FUNCTION_BLOCK "FU SEW DFE32B - PN_REL"	// FB 6119
TITLE = Control of SEW frequency converter with DFE32B via Profinet
//Building:
//Date         Editor                                                     Version
//--------------------------------------------------------------------------------
//31.08.10     A.Kremer (kal)                                            01.00.00
//
//Modifications:
//No. Date     Edit  Description                                    Index Version
//--------------------------------------------------------------------------------
//01  24.04.12 sra   Anpassung zur Integration als Standardbaustein (001) 01.01.00
//02  23.11.15 kst   Anpassung allgemein                            (002) 01.02.00
//03  17.02.16 sra   out_FB_Fehlermeldung = INT                     (003) 01.02.01
//________________________________________________________________________________
//Functional description:
//
//The function cummunicates to a SEW frequency converter MOVITRAC B via Profinet
//interface DFE32B.
//
//Hardwareconfiguration:
//Install GSDML file in hardware catalogue:
// GSDML-V2.1-SEW-DFE-DFS-2Ports-20070426.xml (Internet: www.SEW-EURODRIVE.de)
//
//After the installation you can find the Profinet module  "SEW Gateway DFE32B 
//V1.2" in the hardware catalogue under the menu: "Profinet IO -> other FIELD 
//DEVICES -> Drives -> SEW -> DFE/DFS (2Ports) ->"
//
//Insert this module to the hardware and configurate the following module
//     Slot 1: Empty
//from Slot 2: AS 1 Antrieb (1x3PD)   as often as the number of freq.converter    
// 
//
//
//!!! The nominal motor frequency, motor speed and the nominal motor current must 
//    be transferred to ensure the block functions correctly.
//
//
//Settings at DFE32B:
//
//1. Set IP address via Software: 
//
//2. Execute auto setup at DFE32B by setting DIP switch 2 (AS) to ON
//   All FCs must be switched on and the SBus address set
//   With the auto setup function (DIP switch "AS") it is possible to set up 
//   DFE32B as the gateway without a PC. The function is executed once when the 
//   DIP switch is switched on. The DIP switch must then remain on. The function 
//   can be executed again by switching the DIP switch off and on again.
//
//Frequency converter settings
//
//1. P100 Set setpoint source to SBUS -> value = 10
//
//2. P101 Set control source to SBus -> value 3
//
//3. P301 Set minimum speed in rpm (master value = 15)
//
//4. P302 Set maximum speed in rpm (factory setting = 1500)
//
//5. P303 Set current limit (in % of FC nominal current)
//   (Factory setting =150%)
//
//6. P320 Set automatic motor matching to on (standard setting)
//   (to gauge the motor at start)
//
//7. P500 Switch on speed monitoring
//   (in the case of fault messages P501 increase speed monitoring delay time)
//
//8. P601, P603 and P608 Set binary inputs to ""no function" (=0)
//   Set P602 to 1 = enable (factory setting) DI03 must be bypassed
//
//9. P604 for operation with PTC resistor set to 26 (TF message) otherwise
//   .... zeroing.
//   
//11. P881 Set SBus address of respective frequency converter (from 1 in
//    ascending order)
//
//12. P883 Bus monitoring time -> 5 [s]
//
//13. P884 Check SBus baud rate -> value 500/500 kBaud
//
//14. P870-P872 Setpoint description PA1-PA3
//       P870 = control word 1
//       P871 = speed
//       P872 = reserve
//    P873-P876 Actual value description PE1-PE3
//       P873 = status word 1
//       P874 = speed
//       P875 = output current in % of nominal current
//
AUTHOR : kal
FAMILY : AZO
NAME : standard
VERSION : 0.0
VAR_INPUT
  in_PEA_Adresse : INT ;	//Basisadresse für EA-Daten im PEA-Bereich
  in_FU_Nummer : INT ;	//FU Nummer zur Berechnung des Offsets der Peripherie-EAs
  in_Motordaten_J_N : BOOL ;	//nicht möglich => CLR
  in_Freigabe : BOOL ;	//Steuersignal 1 setzen zum Starten des FUs
  in_Linkslauf : BOOL ;	//Frequenzumformer Linkslauf ein
  in_Quittierung_Stoerung : BOOL ;	//Störung quittieren
  in_Sollfrequenz : REAL ;	//Sollfrequenz in Hz
  in_Motorleistungsfaktor : REAL ;	//nicht vorhanden => 0
  in_Motornennfrequenz : REAL ;	//Wertebereich: 0 - 100 Hz
  in_Motornenndrehzahl : REAL ;	//Wertebereich: 0 - 10000 U/min
  in_Motornennstrom : REAL ;	//Wertebereich: 0- ... A
  in_Motornennspannung : REAL ;	//nicht vorhanden => 0
  in_Motornennleistung : REAL ;	//nicht vorhanden => 0
END_VAR
VAR_OUTPUT
  out_Istfrequenz : REAL ;	//Istfrequenz in Hz
  out_Istdrehzahl : REAL ;	//Istdrehzahl in U/min
  out_Leistung : REAL ;	//nicht vorhanden => 0
  out_Drehmoment : REAL ;	//nicht vorhanden => 0
  out_Motorspannung : REAL ;	//nicht vorhanden => 0
  out_Ausgangsstrom : REAL ;	//Ausgangsstrom des FU
  out_Stoerung : BOOL ;	//1=Gerätestörung
  out_Warnung : BOOL ;
  out_Sollwert_erreicht : BOOL ;	//zeigt 1 an, wenn Istwert gleich Sollwert ist
  out_laeuft : BOOL ;	//=1 wenn Istdrehzahl > 0
  out_FB_Fehlermeldung : INT ;	//0 = ok ; sonst Fehler_Code_L2Dp
  out_Stoerungsnummer : DINT ;	//Stoerungsnummer, bzw. Betriebszustand wenn keine Störung aktiv
END_VAR
VAR
  reserve : ARRAY  [58 .. 99 ] OF BYTE ;
  Prozessdatenkanal_in : STRUCT 	//Prozesseingangsdaten
   PI1_Statuswort : STRUCT
    Zustand_Fehlercode : BYTE ;
    Endstufe_freigegeben : BOOL ;
    Umrichter_betriebsbereit : BOOL ;
    PA_Daten_freigegeben : BOOL ;
    reserve_3 : BOOL ;
    reserve_4 : BOOL ;
    Stoerung_Warnung : BOOL ;
    reserve_6 : BOOL ;	//0 = 1. Satz; 1 = 2. Satz
    reserve_7 : BOOL ;	//0 = 1. Satz; 1 = 2. Satz
   END_STRUCT ;
   PI2_Istdrehzahl : INT ;
   PI3_Ausgangsstrom : INT ;
  END_STRUCT ;
  Prozessdatenkanal_out : STRUCT 	//Prozessausgangsdaten
   PO1_Steuerwort : STRUCT
    Drehrichtung : BOOL ;	//0 = rechts; 1 = links
    Motorpoti_auf : BOOL ;	//00=11= keine Änderung; 01=Hochlauf, 02=Tieflauf
    Motorpoti_ab : BOOL ;
    Festsollwerte_0 : BOOL ;	//00 = Feldbus
    Festsollwerte_1 : BOOL ;
    Festsollwert_Umschaltung : BOOL ;
    reserve_14 : BOOL ;
    reserve_15 : BOOL ;
    Reglersperre : BOOL ;	//Freigabe = '110', sonst Halt
    Freigabe_Schnellstop : BOOL ;
    Freigabe_Normalhalt : BOOL ;
    reserve_3 : BOOL ;
    reserve_4 : BOOL ;
    reserve_5 : BOOL ;	//0 = 1.Satz; 1 = 2.Satz
    Reset_Stoerung : BOOL ;	//0 = 1.Satz; 1 = 2.Satz
    reserve_7 : BOOL ;
   END_STRUCT ;
   PO2_Solldrehzahl : INT ;	//in %
   PO3_keine_Fkt : INT ;
  END_STRUCT ;
  Datenuebertragung : STRUCT
   Schritt_aktiv : BOOL ;
  END_STRUCT ;
  reserve_1 : ARRAY  [122 .. 137 ] OF BYTE ;
END_VAR
VAR_TEMP
  IO_Adr_Parameterkanal : WORD ;
  IO_Adr_Prozessdatenkanal : WORD ;
  Ret_Val_SFC14_1 : INT ;
  Ret_Val_SFC14_2 : INT ;
  Ret_Val_SFC15_1 : INT ;
  Ret_Val_SFC15_2 : INT ;
  SimFactor : REAL ;	//(001)
  Solldrehzahl_tmp : REAL ;
END_VAR
BEGIN
NETWORK
TITLE = Bausteinende wenn PEA-Adresse = 0
      L     #in_PEA_Adresse;
      L     0;
      ==I;
      BEC;
NETWORK
TITLE = Simulation
//Über die Simulaitonsmerker "M 0.5 Simulation intern" oder "M 0.6 Simulation 
//AVP" 
//wird die Funktion des FUs simuliert:
//- Fehler werden zurückgesetzt
//- Bei Freigabe Istdrehzahl=Solldrehzahl, Betrieb und Solldrehzahl erreicht = 
//True
//(002) Überarbeitung 
      O     "M0.5 SimulationInternal";
      O     "M0.6 SimulationAVP";
      JCN   NSIM;
// <<(002)
      SET;
      R     #out_Stoerung;
      R     #out_Warnung;
// >>(002)
      L     L#0;
      T     #out_Stoerungsnummer;
      A     #in_Freigabe;
      =     #out_laeuft;
      =     #out_Sollwert_erreicht;
      L     #in_Sollfrequenz;
      JC    SIMD;
      L     0.000000e+00;
SIMD: T     #out_Istfrequenz;
// <<(002)
// Faktor berechnen
//     L     #out_Istfrequenz
//     L     #in_Motornennfrequenz
//      /R    
//     T     #SimFactor
// Istdrehzahl
//     L     #in_Motornenndrehzahl
//     L     #SimFactor
//      *R    
//     T     #out_Istdrehzahl
// Istleistung
//     L     #in_Motornennleistung
//     L     #SimFactor
//      *R    
//     T     #out_Leistung
// Istspannung
//     L     #in_Motornennspannung
//     L     #SimFactor
//      *R    
//     T     #out_Motorspannung
// Iststrom
//     L     #in_Motornennstrom
//     L     #SimFactor
//      *R    
//     T     #out_Ausgangsstrom
// >>(002)
      BEU;
NSIM: NOP   0;
NETWORK
TITLE = Daten von FU einlesen
//FU-Daten auslesen mit SFC14
//PEA_Adresse zeigt auf den Anfang des EA-Bereiches.
// 6-Byte Prozessdatenkanal
// <<(002)
      L     #in_FU_Nummer;
      +     -1;
      L     6;	// Länge eines Parameterkanals je FU
      *I;
      L     #in_PEA_Adresse;
      +I;
      T     #IO_Adr_Prozessdatenkanal;	// Daten des jeweiligen FU = PEA-Adresse + 8 Byte + (FU-Nr. - 1) * 6
// >>(002)
      CALL  "DPRD_DAT" (
           LADDR                    := #IO_Adr_Prozessdatenkanal,
           RET_VAL                  := #Ret_Val_SFC14_2,
           RECORD                   := #Prozessdatenkanal_in);
NETWORK
TITLE = Istdrehzahl auswerten
//Istdrehzahl in 0,2 U/min
      L     #Prozessdatenkanal_in.PI2_Istdrehzahl;
      ITD;
      DTR;
      L     5.000000e+00;
      /R;
      T     #out_Istdrehzahl;
NETWORK
TITLE = Istfrequenz auswerten
//Istfrequenz (in Hz) = Istdrehzahl (in 0,2 U/min) / 5 * Nennfrequenz / 
//Nenndrehzahl 
      L     #out_Istdrehzahl;
      L     #in_Motornennfrequenz;
      *R;
      L     #in_Motornenndrehzahl;
      /R;
      T     #out_Istfrequenz;	// in Hz
      L     0.000000e+00;	//  wenn kleiner 0 dann negieren 
      <R;
      JCN   E_IF;
      L     #out_Istfrequenz;
      L     -1.000000e+00;
      *R;
      T     #out_Istfrequenz;
E_IF: NOP   0;
NETWORK
TITLE = Stromwert auswerten
      L     #Prozessdatenkanal_in.PI3_Ausgangsstrom;	// in % des FU-Nennstomes 
      ITD;
      DTR;
      L     1.000000e+03;
      /R;
      L     #in_Motornennstrom;
      *R;
      T     #out_Ausgangsstrom;
NETWORK
TITLE = Betriebsmeldung
      A(;
      L     #out_Istfrequenz;
      L     1.000000e+00;
      >R;
      );
      =     #out_laeuft;
NETWORK
TITLE = Sollwert erreicht
      L     #in_Sollfrequenz;
      L     #out_Istfrequenz;
      -R;
      ABS;
      L     1.000000e+00;
      <R;
      =     #out_Sollwert_erreicht;
NETWORK
TITLE = Störungsbit auswerten
//Störungsbit aus Statuswort auswerten
      AN    #Prozessdatenkanal_in.PI1_Statuswort.Umrichter_betriebsbereit;
      A     #Prozessdatenkanal_in.PI1_Statuswort.Stoerung_Warnung;
      O(;
      L     #out_FB_Fehlermeldung;
      L     0;
      <>I;
      );
      O(;
      L     #out_Stoerungsnummer;
      L     0;
      <>D;
      );
      =     #out_Stoerung;
NETWORK
TITLE = Störung resetten
//Störung resetten
//NW Warnungsbit Verschoben (002)
      A     #in_Quittierung_Stoerung;
      A     #Prozessdatenkanal_in.PI1_Statuswort.Stoerung_Warnung;
      =     #Prozessdatenkanal_out.PO1_Steuerwort.Reset_Stoerung;
NETWORK
TITLE = Gerätezustand / Störungsnummer des Frequenzumformers auslesen
//Gerätezustand wenn Bit Störung/Warnung = 0
//Störungsnummer wenn Bit Störung/Warnung = 1
      L     #Prozessdatenkanal_in.PI1_Statuswort.Zustand_Fehlercode;
      ITD;
      T     #out_Stoerungsnummer;
// Störmeldung nur wenn Bit Störung = 1
      A     #Prozessdatenkanal_in.PI1_Statuswort.Stoerung_Warnung;
      JC    ESTO;
      L     0;
      T     #out_Stoerungsnummer;
ESTO: NOP   0;
NETWORK
TITLE = Freigabebefehl bearbeiten
      CLR;
      =     #Prozessdatenkanal_out.PO1_Steuerwort.Reglersperre;
      SET;
      =     #Prozessdatenkanal_out.PO1_Steuerwort.Freigabe_Schnellstop;
      A     #in_Freigabe;
      =     #Prozessdatenkanal_out.PO1_Steuerwort.Freigabe_Normalhalt;
NETWORK
TITLE = Belegung der restlichen Steuerbits
      CLR;
      =     #Prozessdatenkanal_out.PO1_Steuerwort.reserve_3;
      =     #Prozessdatenkanal_out.PO1_Steuerwort.reserve_4;
      =     #Prozessdatenkanal_out.PO1_Steuerwort.reserve_5;
      =     #Prozessdatenkanal_out.PO1_Steuerwort.reserve_7;
      =     #Prozessdatenkanal_out.PO1_Steuerwort.Motorpoti_auf;
      =     #Prozessdatenkanal_out.PO1_Steuerwort.Motorpoti_ab;
      =     #Prozessdatenkanal_out.PO1_Steuerwort.Festsollwerte_0;
      =     #Prozessdatenkanal_out.PO1_Steuerwort.Festsollwerte_1;
      =     #Prozessdatenkanal_out.PO1_Steuerwort.Festsollwert_Umschaltung;
      =     #Prozessdatenkanal_out.PO1_Steuerwort.reserve_14;
      =     #Prozessdatenkanal_out.PO1_Steuerwort.reserve_15;
NETWORK
TITLE = Solldrehzahl
//Solldrehzahl (in 0,2 HZ) 
//Sollfrequenz (in Hz) * 5 * Nenndrehzahl / Nennfrequenz
//(002) Begrenzung Solldrehzahl auf INT 
//
      L     #in_Sollfrequenz;
      L     #in_Motornenndrehzahl;
      *R;
      L     5.000000e+00;
      *R;
      L     #in_Motornennfrequenz;
      /R;
      T     #Solldrehzahl_tmp;	//(002)
      L     3.276700e+04;	//(002)
      >R;	//(002)
      JCN   SD_1;	//(002)
// maximale Drehzahl ausgeben wenn angeforderte größer als Maximalwert ist
      L     3.276700e+04;	//(002)
      RND;	//(002)
      T     #Prozessdatenkanal_out.PO2_Solldrehzahl;	//(002)
      JU    SD_L;	//(002)
// Drehzahl ausgeben wenn angeforderte kleiner als Maximalwert ist
SD_1: L     #Solldrehzahl_tmp;	//(002)
      RND;	//(002)
      T     #Prozessdatenkanal_out.PO2_Solldrehzahl;	//(002)
SD_L: AN    #in_Linkslauf;	//(002)
      JC    E_SD;	//(002)
      L     #Prozessdatenkanal_out.PO2_Solldrehzahl;
      L     -1;
      *I;
      T     #Prozessdatenkanal_out.PO2_Solldrehzahl;
E_SD: NOP   0;
NETWORK
TITLE = Warnungsbit
// (002) Verschoben + Änderung
      A     #Prozessdatenkanal_in.PI1_Statuswort.Umrichter_betriebsbereit;
      A     #Prozessdatenkanal_in.PI1_Statuswort.Stoerung_Warnung;
      O(;	//(002)
      L     #Solldrehzahl_tmp;	//(002)
      L     3.276700e+04;	//(002)
      >=R;	//(002)
      );	//(002)
      O(;	//(002)
      L     #Solldrehzahl_tmp;	//(002)
      L     -3.276700e+04;	//(002)
      <=R;	//(002)
      );	//(002)
      =     #out_Warnung;
NETWORK
TITLE = Netzwerk für nicht unterstützte Funktionen
//Zur Standardisierung der E/A-Parameter aller FUs
      L     0.000000e+00;
      T     #out_Leistung;
      T     #out_Drehmoment;
      T     #out_Motorspannung;
NETWORK
TITLE = Daten an FU senden
// 6-Byte Prozessdatenkanal
      CALL  "DPWR_DAT" (
           LADDR                    := #IO_Adr_Prozessdatenkanal,
           RECORD                   := #Prozessdatenkanal_out,
           RET_VAL                  := #Ret_Val_SFC15_2);
NETWORK
TITLE = Fehlercode L2Dp in FB_Fehlermeldung
      L     0;
      L     #Ret_Val_SFC14_2;
      <>I;
      JC    Fehl;
      L     0;
      L     #Ret_Val_SFC15_2;
      <>I;
      JC    Fehl;
      L     0;
Fehl: T     #out_FB_Fehlermeldung;
END_FUNCTION_BLOCK

FUNCTION "FC2 Taktgeber_Timernachb" : VOID	// FC 2
TITLE = Taktgeber
//Erstellung:
//Datum        Bearbeiter                                                 Version
//--------------------------------------------------------------------------------
//16.12.97     R.Schaffert (sra)                                          01.00.00
//  
//Änderungen:
//Nr. Datum    Bearb Änderung                                       Marke  Version
//--------------------------------------------------------------------------------
//01  09.03.99 sra   Variabler Takteingang                          ()    01.01.00
//02  18.03.99 sra   Fehlerbeseitigung                              ()    01.01.01
//03  01.04.99 jm    Taktzähler auch bei Dauertakt aktiv            ()    01.01.02
//04  14.04.99 sra   Fehlerbeseitigung                              ()    01.01.03
//05  20.12.00 sra   Taktanz.err. rücksetzen bei Dauertakt          ()    01.01.04
//
//________________________________________________________________________________
//Beschreibung:
//
//Diese Funktion generiert ein beliebiges Taktsignal ohne Verwendung eines Timers.
//Es muß ein Impulssignal der Standardimpulse MB4 angelegt werden das über die 
//Taktmerker der CPU und dem Standardbaustein FC13 generiert wird
//Die Zykluszeit muß dabei kleiner sein als das verwendete Taktsignal / 2
//
//Achtung !
//- Am Parameter "in_Rueckmeldung" darf nicht "true" oder "false" angelegt 
//  werden, sondern es muss dem Ausgangssignal "io_Taktausgang" folgen ! 
//- Bei Angabe von z.B. "in_Sollanzahl_Takte" = 5 wird der Parameter 
//  "io_Taktzaehler" von 0..4 hochgezählt
//
AUTHOR : sra
FAMILY : Takt
NAME : Takt_TN
VERSION : 0.0
VAR_INPUT
  in_Freigabe : BOOL ;	//Freigabe Takt
  in_Rueckmeldung : BOOL ;	//Rueckmeldung z.B. Eingang ein
  in_Start_mit_Impuls : BOOL ;	//Takt mit positivem Impuls starten
  in_Dauertakt : BOOL ;	//Dauertakt ? (1=Ja / 0=Nein)
  in_Impuls : BOOL ;	//Impulseingang Takt
  in_Impulszeit_in_100ms : INT ;	//Impulszeit in 100ms
  in_Impulszeit : REAL ;	//Impulszeit fuer Takt in Sekunden
  in_Pausezeit : REAL ;	//Pausezeit fuer Takt in Sekunden
  in_Sollanzahl_Takte : INT ;	//Sollanzahl Takte wenn nicht Dauertakt
END_VAR
VAR_IN_OUT
  io_Taktausgang : BOOL ;	//Taktausgang
  io_Taktanzahl_erreicht : BOOL ;	//Meldung Taktanzahl erreicht
  io_Zeitzaehler : REAL ;	//Zeitzähler (abgelaufene Zeit)
  io_Taktzaehler : INT ;	//Taktzähler
END_VAR
BEGIN
NETWORK
TITLE = Rücksetzen der Zähler und Merker
//Wenn keine Freigabe mehr anliegt werden die in_out Parameter auf 0 gesetzt.
//
      A     #in_Freigabe;
      JC    Strt;
      L     1.000000e-02;
      T     #io_Zeitzaehler;
      L     0;
      T     #io_Taktzaehler;
      SET;
      R     #io_Taktausgang;
      R     #io_Taktanzahl_erreicht;
      BEU;
NETWORK
TITLE = Dauerimpuls oder Dauerpause
Strt: NOP   0;
      L     #in_Impulszeit;
      L     0.000000e+00;
      ==R;
      R     #io_Taktausgang;
      BEC;
      L     #in_Pausezeit;
      L     0.000000e+00;
      ==R;
      S     #io_Taktausgang;
      BEC;
NETWORK
TITLE = Start Takt mit Impuls
//Wenn der Takt mit einem Impuls gestartet werden soll, wird der Ausgang beim 
//Start des Taktes zunächst auf 1 gesetzt.
//Bedingung: Zeitzähler und Taktzähler müssen 0 sein
      A     #in_Freigabe;
      A     #in_Start_mit_Impuls;
      A(;
      A(;
      L     #io_Zeitzaehler;
      L     1.000000e-02;
      ==R;
      );
      A(;
      L     #io_Taktzaehler;
      L     0;
      ==I;
      );
      O;
      A     #in_Dauertakt;
      A     #io_Taktanzahl_erreicht;
      );
      S     #io_Taktausgang;
NETWORK
TITLE = Taktanzahl erreicht ?
//Abfrage ob Taktanzahl erreicht ist
      L     #io_Taktzaehler;
      L     #in_Sollanzahl_Takte;
      >=I;
      S     #io_Taktanzahl_erreicht;
      A     #in_Dauertakt;
      A     #io_Taktanzahl_erreicht;
      JCN   NCCR;	//No Clock Counter Reset
      L     0;
      T     #io_Taktzaehler;
      SET;
      R     #io_Taktanzahl_erreicht;
NCCR: NOP   0;	//No Clock Counter Reset
NETWORK
TITLE = Impuls-Phase des Taktes
//Erhöhung des Zeitzählers während der Impulsphase
//Ist die Sollzeit erreicht wird der Taktzähler erhöht, der Taktausgang 
//zurückgesetzt und der Zeitzähler wieder auf 0 gesetzt
      AN    #io_Taktausgang;
      JC    P_PH;	// wenn Taktausgang nicht gesetzt ist -> Pausephase 
      A     #in_Rueckmeldung;	// solange keine Rückmeldung -> Zeit läuft nicht
      JC    RM_I;
      L     0.000000e+00;
      T     #io_Zeitzaehler;	// Zeitzähler löschen wenn keine Rückmeldung
      JU    ENDE;
RM_I: NOP   0;
      AN    #in_Impuls;
      JC    IMP0;
      L     #in_Impulszeit_in_100ms;
      ITD;
      DTR;
      L     1.000000e-01;
      *R;
      L     #io_Zeitzaehler;	// Zeitzähler erhöhen
      +R;
      T     #io_Zeitzaehler;
      L     #in_Impulszeit;
      <R;
      JC    IMP0;
      SET;
      R     #io_Taktausgang;
      L     #io_Taktzaehler;
      INC   1;
      T     #io_Taktzaehler;
      L     0.000000e+00;
      T     #io_Zeitzaehler;	// Zeitzähler löschen
IMP0: NOP   0;
NETWORK
TITLE = Pause-Phase des Taktes
//Erhöhung des Zeitzählers während der Pausephase
//Ist die Sollzeit erreicht wird der Taktzähler erhöht, der Taktausgang 
//gesetzt und der Zeitzähler wieder auf 0 gesetzt.
//Ist die Solltaktzahl erreicht erfolgt keine weiter Bearbeitung des Netzwerks
P_PH: O     #io_Taktausgang;
      O     #io_Taktanzahl_erreicht;
      JC    ENDE;	// wenn Taktausgang gesetzt ist -> ENDE
      AN    #in_Rueckmeldung;	// solange Rückmeldung -> Zeit läuft nicht
      JC    RM_P;
      L     0.000000e+00;
      T     #io_Zeitzaehler;	// Zeitzähler löschen wenn keine Rückmeldung
      JU    ENDE;
RM_P: NOP   0;
      AN    #in_Impuls;
      JC    ENDE;
      L     #in_Impulszeit_in_100ms;
      ITD;
      DTR;
      L     1.000000e-01;
      *R;
      L     #io_Zeitzaehler;	// Zeitzähler erhöhen
      +R;
      T     #io_Zeitzaehler;
      L     #in_Pausezeit;
      <R;
      JC    ENDE;
      SET;
      S     #io_Taktausgang;
      L     0.000000e+00;
      T     #io_Zeitzaehler;	// Zeitzähler löschen
ENDE: NOP   0;
END_FUNCTION

FUNCTION "FC3 Timernachbildung" : VOID	// FC 3
TITLE = Ein- / Ausschaltverzögerung
//Erstellung:
//Datum        Bearbeiter                                                 Version
//--------------------------------------------------------------------------------
//27.05.97     R.Schaffert (sra)                                          01.00.00
//  
//Änderungen:
//Nr. Datum    Bearb Änderung                                       Marke  Version
//--------------------------------------------------------------------------------
//01  05.02.1999  hus      Parameter "Reset" eingeführt             ()    01.01.00
//02  22.03.1999  sra      Fehlerbeseitigung                        ()    01.01.01
//03  25.08.1999  jm       SV inkl. Reset (getestet)                ()    01.02.00
//04  27.09.1999  jm       SI inkl. Reset (getestet)                ()    01.03.00
//05  26.05.2002  jm       SZ inkl. Reset (getestet): Zeitzähler    ()    01.04.00
//06  22.05.2007  sra      Zeitzaehler läuft bei SE weiter          (006) 01.04.01
//
//________________________________________________________________________________
//Beschreibung:
//
//Diese Funktion generiert eine Ein- bzw. Ausschaltverzögerung ohne Verwendung 
//eines Timers. 
//
//Es muß ein Impulssignal "in_Impuls" der Standardimpulse MB4 angelegt werden, 
//das durch die Angabe der Taktzeit in 1/100ms "in_Impulszeit_in_100ms" 
//spezifiziert wird.
//
//Wird der Eingang "Reset" gesetzt, wird der Ausgang zurückgesetzt und der 
//Zeitzähler wird auf 0 gesetzt.
//
//SE: Durch Auswahl von "E" als Verzögerungsart wird eine Einschaltverzögerung 
//gestartet sobald "in_Freigabe" vorhanden ist. Der Ausgang "io_Ausgangssignal" 
//wird nach Ablauf der Verzögerungszeit "in_Verzoegerungszeit" auf 1 gesetzt und 
//steht dann solange an bis die Freigabe nicht mehr vorhanden ist. Der Eingang 
//"in_Reset"  bewirkt eine Nullung der Istzeit und ein Rücksetzen des Ausgangs. 
//Wird der Eingang "in_Reset" weggenommen so startet die Verzögerungszeit von 
//vorne, es sei denn "in_Freigabe" ist dann nicht mehr vorhanden.
//
//SA: Durch Auswahl von "A" als Verzögerungsart wird eine Ausschaltverzögerung 
//gestartet sobald "in_Freigabe" vorhanden ist. Der Ausgang wird sofort mit 
//dem Signal "in_Freigabe" auf 1 gesetzt. Sobald die Freigabe nicht mehr 
//vorhanden ist wird die Ausschaltverzögerung gestartet. Der Ausgang 
//"io_Ausgangssignal" steht weiterhin auf 1. Nach Ablauf der Verzögerungszeit 
//"in_Verzoegerungszeit" wird der Ausgang "io_Ausgangssignal" auf 0 gesetzt. Der 
//Eingang "in_Reset" bewirkt eine Nullung der Istzeit und ein Rücksetzen des 
//Ausgangs. Wird der Eingang "in_Reset" weggenommen so startet die Funktion von 
//vorne, es sei denn "in_Freigabe" ist dann nicht mehr vorhanden.
//
//SV: Durch Auswahl von "V" als Verzögerungsart wird ein verlängerter Impuls 
//gestartet sobald "in_Freigabe" vorhanden ist. Der Ausgang "io_Ausgangssignal" 
//wird für die Verzögerungszeit "in_Verzoegerungszeit" auf 1 gesetzt, unabhängig 
//vom Eingang "in_Freigabe". Der Eingang "in_Reset" bewirkt eine Nullung der 
//Istzeit und ein Rücksetzen des Ausgangs. Wird der Eingang "in_Reset" 
//weggenommen so startet der Impuls von vorne, es sei denn "in_Freigabe" ist dann 
//nicht mehr vorhanden.  
//
//SI: Durch Auswahl von "I" als Verzögerungsart wird ein Impuls gestartet sobald 
//"in_Freigabe" vorhanden ist. Der Ausgang "io_Ausgangssignal" wird für die 
//bestimmte Zeit auf 1 gesetzt, abhängig vom Eingang "in_Freigabe". Der Eingang 
//"Reset" bewirkt eine Nullung der Istzeit und ein Rücksetzen des Ausgangs 
//"io_Ausgangssignal". Wird der Eingang "Reset" weggenommen so startet der Impuls 
//von vorne, es sei denn "in_Freigabe" ist dann nicht mehr vorhanden.
//
//SZ: Diese Funktion kann als Zeitzähler bezeichnet werden. Sobald "in_Freigabe" 
//vorhanden ist wird die Zeit hochgezählt. Ohne "in_Freigabe" bleibt die Zeit 
//stehen, sobald "in_Freigabe" wieder vorhanden ist wird weiter gezählt. Ist die 
//Sollzeit "in_Verzoegerungszeit" erreicht und "in_Freigabe" geht weg, wird der 
//Zeitzähler rückgesetzt. Der Eingang "Reset" bewirkt eine Nullung der Istzeit 
//und ein Rücksetzen des Ausgangs "io_Ausgangssignal". Wird der Eingang "Reset" 
//weggenommen so startet der Zeitzähler von vorne, es sei denn "in_Freigabe" ist 
//dann nicht mehr vorhanden.
AUTHOR : hus
FAMILY : AZO
VERSION : 0.1
VAR_INPUT
  in_Freigabe : BOOL ;	//Freigabe Timernachbildung
  in_Reset : BOOL ;	//Reset (z.B. Steuerspannung aus)
  in_Impuls : BOOL ;	//Impulseingang (M1.7)
  in_Impulszeit_in_100ms : INT ;	//Impulszeit in 100ms (MW6)
  in_Verzoegerungsart : CHAR ;	//'E'=Einschalt-,'A'=Ausschaltverz.,'V'=verl.Impuls,'I'= Impuls,'Z'=Zeitzähler
  in_Verzoegerungszeit : REAL ;	//Verzögerungszeit in Sekunden
END_VAR
VAR_IN_OUT
  io_Ausgangssignal : BOOL ;	//Timerausgang
  io_Zeitzaehler : REAL ;	//Zeitzähler (abgelaufene Zeit)
END_VAR
BEGIN
NETWORK
TITLE = Einschaltverzögerung
//Einschaltverzögerung
      L     #in_Verzoegerungsart;
      L     'E';
      <>I;
      JC    E1;
      A     #in_Freigabe;
      JC    SE;
      SET;
      R     #io_Ausgangssignal;
      L     0.000000e+00;
      T     #io_Zeitzaehler;
      JU    E1;
//    O     #io_Ausgangssignal // (006)
SE:   ON    #in_Impuls;
      JC    E1;
      L     #in_Impulszeit_in_100ms;
      ITD;
      DTR;
      L     1.000000e-01;
      *R;
      L     #io_Zeitzaehler;
      +R;
      T     #io_Zeitzaehler;
      L     #in_Verzoegerungszeit;
      >=R;
      S     #io_Ausgangssignal;
E1:   NOP   0;
NETWORK
TITLE = Ausschaltverzögerung
//Ausschaltverzögerung
      L     #in_Verzoegerungsart;
      L     'A';
      <>I;
      JC    E2;
      AN    #in_Freigabe;
      JC    SA;
      SET;
      S     #io_Ausgangssignal;
      L     0.000000e+00;
      T     #io_Zeitzaehler;
      JU    E2;
SA:   ON    #io_Ausgangssignal;
      ON    #in_Impuls;
      JC    E2;
      L     #in_Impulszeit_in_100ms;
      ITD;
      DTR;
      L     1.000000e-01;
      *R;
      L     #io_Zeitzaehler;
      +R;
      T     #io_Zeitzaehler;
      L     #in_Verzoegerungszeit;
      >=R;
      R     #io_Ausgangssignal;
E2:   NOP   0;
NETWORK
TITLE = Verlängerter Impuls
//Verlängerter Impuls
      L     #in_Verzoegerungsart;
      L     'V';
      <>I;
      JC    E3;
      O     #in_Freigabe;
      O     #io_Ausgangssignal;
      JC    SV;
      CLR;
      =     #io_Ausgangssignal;
      L     0.000000e+00;
      T     #io_Zeitzaehler;
      JU    E3;
SV:   A     #in_Freigabe;
      S     #io_Ausgangssignal;
      L     #io_Zeitzaehler;
      L     #in_Verzoegerungszeit;
      >=R;
      R     #io_Ausgangssignal;
      ON    #in_Impuls;
      ON    #io_Ausgangssignal;
      JC    E3;
      L     #in_Impulszeit_in_100ms;
      ITD;
      DTR;
      L     1.000000e-01;
      *R;
      L     #io_Zeitzaehler;
      +R;
      T     #io_Zeitzaehler;
      L     #in_Verzoegerungszeit;
      >=R;
      R     #io_Ausgangssignal;
E3:   NOP   0;
NETWORK
TITLE = Impuls
//Impuls
      L     #in_Verzoegerungsart;
      L     'I';
      <>I;
      JC    E4;
      A     #in_Freigabe;
      JC    SI;
      CLR;
      =     #io_Ausgangssignal;
      L     0.000000e+00;
      T     #io_Zeitzaehler;
      JU    E4;
SI:   A     #in_Freigabe;
      S     #io_Ausgangssignal;
      L     #io_Zeitzaehler;
      L     #in_Verzoegerungszeit;
      >=R;
      R     #io_Ausgangssignal;
      ON    #in_Impuls;
      ON    #io_Ausgangssignal;
      JC    E4;
      L     #in_Impulszeit_in_100ms;
      ITD;
      DTR;
      L     1.000000e-01;
      *R;
      L     #io_Zeitzaehler;
      +R;
      T     #io_Zeitzaehler;
      L     #in_Verzoegerungszeit;
      >=R;
      R     #io_Ausgangssignal;
E4:   NOP   0;
NETWORK
TITLE = Zeitzähler 'Z'
//Einschaltverzögerung
      L     #in_Verzoegerungsart;
      L     'Z';
      <>I;
      JC    E5;
      AN    #in_Freigabe;
      A     #io_Ausgangssignal;
      JCN   SZ;	// Zeitzähler wird gelöscht, wenn Zeit abgelaufen und FRG weg geht
      SET;
      R     #io_Ausgangssignal;
      L     0.000000e+00;
      T     #io_Zeitzaehler;
      JU    E5;
SZ:   O     #io_Ausgangssignal;
      ON    #in_Freigabe;
      ON    #in_Impuls;
      JC    E5;
      L     #in_Impulszeit_in_100ms;
      ITD;
      DTR;
      L     1.000000e-01;
      *R;
      L     #io_Zeitzaehler;
      +R;
      T     #io_Zeitzaehler;
      L     #in_Verzoegerungszeit;
      >=R;
      S     #io_Ausgangssignal;
E5:   NOP   0;
NETWORK
TITLE = Rücksetzen Ausschaltverzögerung wenn Reseteingang = "True". 
      AN    #in_Reset;
      JC    E6;
      A     #io_Ausgangssignal;
      R     #io_Ausgangssignal;
      L     0.000000e+00;
      T     #io_Zeitzaehler;
E6:   NOP   0;
END_FUNCTION

FUNCTION "FC4 Blocktransfer ANY-Q" : VOID	// FC 4
TITLE = BlockTransfer mit ANY-Zeiger als Quelle
//Erstellung:
//Datum        Bearbeiter                                                Version
//--------------------------------------------------------------------------------
//09.03.99     R.Schaffert (sra)                                         V01.00.00
//
//Änderungen:
//Nr. Datum    Bearb Beschreibung                                   Marke Version
//--------------------------------------------------------------------------------
//01 30.06.99  sra   Fehlerbeseitigung                                    01.00.01
//02 27.01.04  gea   Fehlerbeseitigung Quell-DW > 8192              (002) 01.00.02
//03 13.12.05  sra   Fehlerbeseitigung Ziel-DW > 8192               (003) 01.00.03
//04 10.06.10  sra   Bereich > 32767 kopieren                       (004) 01.00.04
//________________________________________________________________________________
//Funktion:
//
//Blocktranferfunktion mit Systemfunktion SFC20
//-Bei "in_Ziel_Typ" = 'E' werden die Aktualwerte des in "in Quelle" definierten 
// Bereiches an den durch "in_Ziel_DW" definierten Eingangsbereich kopiert.
//-Bei "in_Ziel_Typ" = 'A' werden die Aktualwerte des in "in Quelle" definierten 
// Bereiches an den durch "in_Ziel_DW" definierten Ausgangsbereich kopiert.
//-Bei "in_Ziel_Typ" = 'M' werden die Aktualwerte des in "in Quelle" definierten 
// Bereiches an den durch "in_Ziel_DW" definierten Merkerbereich kopiert.
//-Bei "in_Ziel_Typ" = 'D' werden die Aktualwerte des in "in Quelle" definierten 
// Bereiches an den durch "in_Ziel_DB" und "in_Ziel_DW" definierten 
// Global-Datenbaustein kopiert.
//-Bei "in_Ziel_Typ" = 'I' werden die Aktualwerte des in "in Quelle" definierten 
// Bereiches an den durch "in_Ziel_DW" definierten Zielbereich des aktuellen 
// Instanz-Datenbausteines kopiert.
//
//An diesen Funktionsbaustein und den SFC20 werden Zeiger (ANY-Zeiger) angelegt, 
//die die Datenquelle definieren. Zeiger ist folgendermaßen aufgebaut:
//     Byte n       B#16#10 
//     Byte n+1     Datentyp (Bool, Byte, usw.)
//     Byte n+2     Anzahl der Datentypen die kopiert werdn sollen (2 Byte)
//     Byte n+4     Datenbausteinnummer (2 Byte)
//     Byte n+6     Bereichszeiger (4 Byte)
//
//Aufbau des bereichsübergreifenden Zeigers:  10000ZZZ 00000yyy yyyyyyyy yyyyyxxx
//      z = Operandenbereich (codiert)
//      y = Byte-Adresse
//      x = Bit-Adresse
//
AUTHOR : sra
FAMILY : AZO
VERSION : 0.0
VAR_INPUT
  in_Quelle : ANY ;	//ANY-Zeiger auf Quelle
  in_Ziel_Typ : CHAR ;	//E=Eingang, A=Ausgang, M=Merker, D=DB, I=Instanz-DB
  in_Ziel_DB : INT ;	//Ziel-DB bei DW-Transfer
  in_Ziel_DW : INT ;	//Ziel-DW Byte-Adresse des Ziels
END_VAR
VAR_OUTPUT
  out_Fehler : INT ;	//1=Ziel-Typ ungültig, 2=DB existiert nicht, 3= DB zu kurz, SFC20 Fehlermeldung
END_VAR
VAR_TEMP
  Quellzeiger : ANY ;
  Zielzeiger : ANY ;
  Quell_DB : INT ;
  Quell_DW : INT ;
  Blocklaenge : INT ;
  Datentyp : BYTE ;
  SFC20_return : INT ;
  Operandenbereich : INT ;
  DB_Test_Nr : WORD ;
  DB_Test_Fehler : INT ;
  DB_Test_Anz_Byte : WORD ;
  DB_Test_Schreib_Schutz : BOOL ;
END_VAR
BEGIN
NETWORK
TITLE = Operandenbereich Quelle codieren
//Bereichscodierung für Quelltyp durchführen
//Operandenbereich im bereichsübergreifenden Zeiger
//
//Aufbau des bereichsübergreifenden Zeigers:  10000ZZZ 00000yyy yyyyyyyy yyyyyxxx
//      z = Operandenbereich (codiert)
//      y = Byte-Adresse
//      x = Bit-Adresse
//    
      L     P##in_Quelle;
      LAR1;
      L     B [AR1,P#1.0];
      T     #Datentyp;
      L     W [AR1,P#2.0];
      T     #Blocklaenge;
      L     W [AR1,P#4.0];
      T     #Quell_DB;
      L     D [AR1,P#6.0];
      L     DW#16#FFFFFF;
      AD;
      SRD   3;	//(002)
      T     #Quell_DW;
      L     D [AR1,P#6.0];
      L     DW#16#F000000;
      AD;
      SRD   24;
      T     #Operandenbereich;
NETWORK
TITLE = Quell-Datenbaustein prüfen
//Überprüfen bei Quelltyp = D,I : Baustein existiert und ist ausreichend lang
      L     #Operandenbereich;
      L     5;	//Quelle ist Instanz-DB 
      <>I;
      JC    M004;
      L     DINO;	//Nummer akt. Instanz-DB
      T     #Quell_DB;
      T     #DB_Test_Nr;
      JU    M005;
M004: L     #Operandenbereich;
      L     4;	//Quelle ist Global-DB
      <>I;
      JC    M003;
      L     #Quell_DB;
      T     #DB_Test_Nr;
M005: CALL  "TEST_DB" (
           DB_NUMBER                := #DB_Test_Nr,
           RET_VAL                  := #DB_Test_Fehler,
           DB_LENGTH                := #DB_Test_Anz_Byte,
           WRITE_PROT               := #DB_Test_Schreib_Schutz);
      L     #DB_Test_Fehler;
      L     0;
      ==I;
      JC    M006;
      L     2;	//DB existiert nicht
      T     #out_Fehler;
      BEU;
M006: L     #Quell_DW;
      L     #Blocklaenge;
      +D;	// (004)
      L     #DB_Test_Anz_Byte;
      <=D;	// (004)
      JC    M003;
      L     3;	//DB nicht ausreichend lang
      T     #out_Fehler;
      BEU;
M003: NOP   0;
NETWORK
TITLE = Quellezeiger belegen
//Quelle vom Typ "ANY" erstellen
      LAR1  P##Quellzeiger;
      L     B#16#10;
      T     LB [AR1,P#0.0];	//Syntax-ID ist immer 10h bei AWL
      L     #Datentyp;
      T     LB [AR1,P#1.0];	// Datentyp 
      L     #Blocklaenge;
      T     LW [AR1,P#2.0];	// Anzahl der Bytes die kopiert werden sollen
      L     #Quell_DB;
      T     LW [AR1,P#4.0];	// Datenbaustzeinnummer
      L     #Operandenbereich;
      L     128;	// 128 addieren (Bit 31 muß 1 sein)
      +I;
      SLD   24;	// 24 Stellen nach links schieben
      L     #Quell_DW;
      SLD   3;	// Quell-DW an Byte-Adresse schieben   //(002)
      +D;	// Zeiger zusammenfügen
      T     LD [AR1,P#6.0];	// siehe Aufbau Bereichszeiger NW1
NETWORK
TITLE = Operandenbereich Ziel codieren
//Bereichscodierung für Zieltyp durchführen
//Operandenbereich im bereichsübergreifenden Zeiger
//
//Aufbau des bereichsübergreifenden Zeigers:  10000ZZZ 00000yyy yyyyyyyy yyyyyxxx
//      z = Operandenbereich (codiert)
//      y = Byte-Adresse
//      x = Bit-Adresse
//    
      L     #in_Ziel_Typ;
      L     'E';	// Ziel = Eingänge
      ==I;
      L     1;
      JC    M002;
      L     #in_Ziel_Typ;
      L     'A';	// Ziel = Ausgänge
      ==I;
      L     2;
      JC    M002;
      L     #in_Ziel_Typ;
      L     'M';	// Ziel = Merker
      ==I;
      L     3;
      JC    M002;
      L     #in_Ziel_Typ;
      L     'D';	// Ziel = DB (Globaldaten)
      ==I;
      L     4;
      JC    M002;
      L     #in_Ziel_Typ;
      L     'I';	// Ziel = Instanz-DB
      ==I;
      L     5;
      JC    M002;
      L     #in_Ziel_Typ;
      L     'L';	// Ziel = Temporäre-Lokal-Daten
      ==I;
      L     6;
      JC    M002;
      L     #in_Ziel_Typ;
      L     'V';	// Ziel = temp. Lokaldaten des Vorgängerbausteins
      ==I;
      L     7;
      JC    M002;
      L     1;	// Kein gültiger Parameter -> Fehler und Ende
      T     #out_Fehler;
      BEU;
M002: T     #Operandenbereich;
NETWORK
TITLE = Ziel-Datenbaustein prüfen
//Überprüfen bei Zieltyp = D,I : Baustein existiert und ist ausreichend lang
      L     #Operandenbereich;
      L     5;	//Ziel ist Instanz-DB 
      <>I;
      JC    M007;
      L     DINO;	//Nummer akt. Instanz-DB
      T     #in_Ziel_DB;
      T     #DB_Test_Nr;
      JU    M008;
M007: L     #Operandenbereich;
      L     4;	//Ziel ist Global-DB
      <>I;
      JC    M010;
      L     #in_Ziel_DB;
      T     #DB_Test_Nr;
M008: CALL  "TEST_DB" (
           DB_NUMBER                := #DB_Test_Nr,
           RET_VAL                  := #DB_Test_Fehler,
           DB_LENGTH                := #DB_Test_Anz_Byte,
           WRITE_PROT               := #DB_Test_Schreib_Schutz);
      L     #DB_Test_Fehler;
      L     0;
      ==I;
      JC    M009;
      L     2;	//DB existiert nicht
      T     #out_Fehler;
      BEU;
M009: L     #in_Ziel_DW;
      L     #Blocklaenge;
      +D;	// (004)
      L     #DB_Test_Anz_Byte;
      <=D;	// (004)
      JC    M010;
      L     3;	//DB nicht ausreichend lang
      T     #out_Fehler;
      BEU;
M010: NOP   0;
NETWORK
TITLE = Zielzeiger belegen
//Ziel vom Typ "ANY" erstellen
      LAR1  P##Zielzeiger;
      L     B#16#10;
      T     LB [AR1,P#0.0];	//Syntax-ID ist immer 10h bei AWL
      L     #Datentyp;
      T     LB [AR1,P#1.0];	// Datentyp 
      L     #Blocklaenge;
      T     LW [AR1,P#2.0];	// Anzahl der Bytes die kopiert werden sollen
      L     #in_Ziel_DB;
      T     LW [AR1,P#4.0];	// Datenbaustzeinnummer
      L     #Operandenbereich;
      L     128;	// 128 addieren (Bit 31 muß 1 sein)
      +I;
      SLD   24;	// 24 Stellen nach links schieben
      L     #in_Ziel_DW;
      SLD   3;	// Quell-DW an Byte-Adresse schieben (003)
      +D;	// Zeiger zusammenfügen
      T     LD [AR1,P#6.0];	// siehe Aufbau Bereichszeiger NW1
NETWORK
TITLE = Blocktransfer
//Blocktransfer mit Systemfunktion SFC20
      CALL  "BLKMOV" (
           SRCBLK                   := #Quellzeiger,
           RET_VAL                  := #SFC20_return,
           DSTBLK                   := #Zielzeiger);
NETWORK
TITLE = Rückgabewert SFC20
//Rückgabewert des SFC20 übergeben
      L     #SFC20_return;
      T     #out_Fehler;
END_FUNCTION

FUNCTION "FC5 Blocktransfer" : VOID	// FC 5
TITLE = BlockTransfer
//Erstellung:
//Datum        Bearbeiter                                                 Version
//--------------------------------------------------------------------------------
//26.06.97     G.Herkert (hkt)                                            01.00.00
//
//Änderungen:
//Nr. Datum    Bearb Beschreibung                                   Marke Version
//--------------------------------------------------------------------------------
//01  20.05.98 sra   komplette Überarbeitung                              02.00.00
//02  29.10.98 gea   Überprüfung Länge und Existenz DBs                   02.01.00
//03  24.11.98 gea   'I' kopiert in/von akt Instanz-DB                    02.02.00
//04  10.05.99 sra   Bereichszeigerberechnung korrigiert                  02.02.01
//05  10.12.01 gea   'K' löscht Bereich                             (005) 02.03.00
//06  07.06.10 sra   Bereich > 32767 kopieren                       (006) 02.03.01
//
//________________________________________________________________________________
//Funktion:
//
//Blocktranferfunktion mit Systemfunktion SFC20
//-Bei "Quell_Typ" = 'E' werden die Aktualwerte der in "Quell_DW" definierten 
// Eingangsadressen ausgelesen und kopiert.
//-Bei "Quell_Typ" = 'A' werden die Aktualwerte der in "Quell_DW" definierten 
// Ausgangsadressen ausgelesen und kopiert.
//-Bei "Quell_Typ" = 'M' werden die Aktualwerte der in "Quell_DW" definierten 
// Merkeradressen ausgelesen und kopiert.
//-Bei "Quell_Typ" = 'D' werden die Aktualwerte der in "Quell-DB" und "Quell_DW"  
// definierten Datenworte ausgelesen und kopiert.
//-Bei "Quell_Typ" = 'I' werden die Aktualwerte der in "Quell_DW" definierten 
// Datenworte des aktuellen Instanz-DBs ausgelesen und kopiert.
//
//-Bei "Ziel_Typ" = 'E' werden die definierten Quelldaten an den durch 
// "in_Ziel_DW" definierten Eingangsbereich kopiert.
//-Bei "Ziel_Typ" = 'A' werden die definierten Quelldaten an den durch 
// "in_Ziel_DW" definierten Ausgangsbereich kopiert.
//-Bei "Ziel_Typ" = 'M' werden die definierten Quelldaten an den durch 
// "in_Ziel_DW" definierten Merkerbereich kopiert.
//-Bei "Ziel_Typ" = 'D' werden die definierten Quelldaten an den durch  
//"in_Ziel_DB" und "in_Ziel_DW" definierten Global-Datenbaustein kopiert.
//-Bei "Ziel_Typ" = 'I' werden die definierten Quelldaten an den durch  
// "in_Ziel_DW" definierten Zielbereich des aktuellen Instanz-Datenbausteines  
// kopiert.
//
//An den SFC20 werden Zeiger (ANY-Zeiger) angelegt die die Quelle und das Ziel 
//beschreiben. Zeiger sind folgendermaßen aufgebaut:
//     Byte n       B#16#10 
//     Byte n+1     Datentyp (Bool, Byte, usw.)
//     Byte n+2     Anzahl der Datentypen die kopiert werdn sollen (2 Byte)
//     Byte n+4     Datenbausteinnummer (2 Byte)
//     Byte n+6     Bereichszeiger (4 Byte)
//
//Aufbau des bereichsübergreifenden Zeigers:  10000ZZZ 00000yyy yyyyyyyy yyyyyxxx
//      z = Operandenbereich (codiert)
//      y = Byte-Adresse
//      x = Bit-Adresse
AUTHOR : hkt
FAMILY : AZO
VERSION : 0.0
VAR_INPUT
  Quell_Typ : CHAR ;	//E=Eingang, A=Ausgang, M=Merker, D=DB, I=Instanz-DB, K=Löschen
  Quell_DB : INT ;	//Quell-Datenbaustein bei DW-Transfer
  Quell_DW : INT ;	//Quell-Datenwort, Byte-Adresse der Quelle
  Ziel_Typ : CHAR ;	//E=Eingang, A=Ausgang, M=Merker, D=DB, I=Instanz-DB
  Ziel_DB : INT ;	//Ziel-Datenbaustein bei DW-Transfer
  Ziel_DW : INT ;	//Ziel-Datenwort, Byte-Adresse des Zieles
  Block_Laenge : INT ;	//Blocklänge in Byte
END_VAR
VAR_OUTPUT
  outFehler : INT ;	//1=Ziel-Typ ungültig, 2=DB existiert nicht, 3= DB zu kurz, SFC20 Fehlermeldung
END_VAR
VAR_TEMP
  Quellzeiger : ANY ;
  Zielzeiger : ANY ;
  SFC20_return : INT ;
  Operandenbereich : INT ;
  DB_Test_Nr : WORD ;
  DB_Test_Fehler : INT ;
  DB_Test_Anz_Byte : WORD ;
  DB_Test_Schreib_Schutz : BOOL ;
END_VAR
BEGIN
NETWORK
TITLE = Bereich in DB-löschen
//(005)
      A(;
      L     #Quell_Typ;
      L     'K';
      ==I;
      );
      A(;
      L     #Ziel_Typ;
      L     'D';
      ==I;
      );
      JCN   BLOE;
      CALL  "FC30 DB vorbelegen" (
           DB_Nr                    := #Ziel_DB,
           DW_Anfang                := #Ziel_DW,
           Anzahl_Bytes             := #Block_Laenge,
           Wert                     := 0);
      BEU;
BLOE: NOP   0;
NETWORK
TITLE = Operandenbereich Quelle codieren
//Bereichscodierung für Quelltyp durchführen
//Operandenbereich im bereichsübergreifenden Zeiger
//
//Aufbau des bereichsübergreifenden Zeigers:  10000ZZZ 00000yyy yyyyyyyy yyyyyxxx
//      z = Operandenbereich (codiert)
//      y = Byte-Adresse
//      x = Bit-Adresse
//    
      L     #Quell_Typ;
      L     'E';	// Quelle = Eingänge
      ==I;
      L     1;
      JC    M001;
      L     #Quell_Typ;
      L     'A';	// Quelle = Ausgänge
      ==I;
      L     2;
      JC    M001;
      L     #Quell_Typ;
      L     'M';	// Quelle = Merker
      ==I;
      L     3;
      JC    M001;
      L     #Quell_Typ;
      L     'D';	// Quelle = DB (Globaldaten)
      ==I;
      L     4;
      JC    M001;
      L     #Quell_Typ;
      L     'I';	// Quelle = Instanz-DB
      ==I;
      L     5;
      JC    M001;
      L     #Quell_Typ;
      L     'L';	// Quelle = Temporäre-Lokal-Daten
      ==I;
      L     6;
      JC    M001;
      L     #Quell_Typ;
      L     'V';	// Quelle = temp. Lokaldaten des Vorgängerbausteins
      ==I;
      L     7;
      JC    M001;
      L     1;	// Kein gültiger Parameter -> Fehler und Ende
      T     #outFehler;
      BEU;
M001: T     #Operandenbereich;
NETWORK
TITLE = Quell-Datenbaustein prüfen
//Überprüfen bei Quelltyp = D,I : Baustein existiert und ist ausreichend lang
      L     #Operandenbereich;
      L     5;	//Quelle ist Instanz-DB 
      <>I;
      JC    M004;
      L     DINO;	//Nummer akt. Instanz-DB
      T     #Quell_DB;
      T     #DB_Test_Nr;
      JU    M005;
M004: L     #Operandenbereich;
      L     4;	//Quelle ist Global-DB
      <>I;
      JC    M003;
      L     #Quell_DB;
      T     #DB_Test_Nr;
M005: CALL  "TEST_DB" (
           DB_NUMBER                := #DB_Test_Nr,
           RET_VAL                  := #DB_Test_Fehler,
           DB_LENGTH                := #DB_Test_Anz_Byte,
           WRITE_PROT               := #DB_Test_Schreib_Schutz);
      L     #DB_Test_Fehler;
      L     0;
      ==I;
      JC    M006;
      L     2;	//DB existiert nicht
      T     #outFehler;
      BEU;
M006: L     #Quell_DW;
      L     #Block_Laenge;
      +D;	// (006)    
      L     #DB_Test_Anz_Byte;
      <=D;	// (006)    
      JC    M003;
      L     3;	//DB nicht ausreichend lang
      T     #outFehler;
      BEU;
M003: NOP   0;
NETWORK
TITLE = Quellezeiger belegen
//Quelle vom Typ "ANY" erstellen
      LAR1  P##Quellzeiger;
      L     B#16#10;
      T     LB [AR1,P#0.0];	//Syntax-ID ist immer 10h bei AWL
      L     2;
      T     LB [AR1,P#1.0];	// Datentyp = 2 (Byte)
      L     #Block_Laenge;
      T     LW [AR1,P#2.0];	// Anzahl der Bytes die kopiert werden sollen
      L     #Quell_DB;
      T     LW [AR1,P#4.0];	// Datenbaustzeinnummer
      L     #Operandenbereich;
      L     128;	// 128 addieren (Bit 31 muß 1 sein)
      +I;
      SLD   24;	// 24 Stellen nach rechts schieben
      L     #Quell_DW;
      SLD   3;	// Quell-DW an Byte-Adresse schieben 
      +D;	// Zeiger zusammenfügen
      T     LD [AR1,P#6.0];	// siehe Aufbau Bereichszeiger NW1
NETWORK
TITLE = Operandenbereich Ziel codieren
//Bereichscodierung für Zieltyp durchführen
//Operandenbereich im bereichsübergreifenden Zeiger
//
//Aufbau des bereichsübergreifenden Zeigers:  10000ZZZ 00000yyy yyyyyyyy yyyyyxxx
//      z = Operandenbereich (codiert)
//      y = Byte-Adresse
//      x = Bit-Adresse
//    
      L     #Ziel_Typ;
      L     'E';	// Ziel = Eingänge
      ==I;
      L     1;
      JC    M002;
      L     #Ziel_Typ;
      L     'A';	// Ziel = Ausgänge
      ==I;
      L     2;
      JC    M002;
      L     #Ziel_Typ;
      L     'M';	// Ziel = Merker
      ==I;
      L     3;
      JC    M002;
      L     #Ziel_Typ;
      L     'D';	// Ziel = DB (Globaldaten)
      ==I;
      L     4;
      JC    M002;
      L     #Ziel_Typ;
      L     'I';	// Ziel = Instanz-DB
      ==I;
      L     5;
      JC    M002;
      L     #Ziel_Typ;
      L     'L';	// Ziel = Temporäre-Lokal-Daten
      ==I;
      L     6;
      JC    M002;
      L     #Ziel_Typ;
      L     'V';	// Ziel = temp. Lokaldaten des Vorgängerbausteins
      ==I;
      L     7;
      JC    M002;
      L     1;	// Kein gültiger Parameter -> Fehler und Ende
      T     #outFehler;
      BEU;
M002: T     #Operandenbereich;
NETWORK
TITLE = Ziel-Datenbaustein prüfen
//Überprüfen bei Zieltyp = D,I : Baustein existiert und ist ausreichend lang
      L     #Operandenbereich;
      L     5;	//Ziel ist Instanz-DB 
      <>I;
      JC    M007;
      L     DINO;	//Nummer akt. Instanz-DB
      T     #Ziel_DB;
      T     #DB_Test_Nr;
      JU    M008;
M007: L     #Operandenbereich;
      L     4;	//Ziel ist Global-DB
      <>I;
      JC    M010;
      L     #Ziel_DB;
      T     #DB_Test_Nr;
M008: CALL  "TEST_DB" (
           DB_NUMBER                := #DB_Test_Nr,
           RET_VAL                  := #DB_Test_Fehler,
           DB_LENGTH                := #DB_Test_Anz_Byte,
           WRITE_PROT               := #DB_Test_Schreib_Schutz);
      L     #DB_Test_Fehler;
      L     0;
      ==I;
      JC    M009;
      L     2;	//DB existiert nicht
      T     #outFehler;
      BEU;
M009: L     #Ziel_DW;
      L     #Block_Laenge;
      +D;	// (006)    
      L     #DB_Test_Anz_Byte;
      <=D;	// (006)    
      JC    M010;
      L     3;	//DB nicht ausreichend lang
      T     #outFehler;
      BEU;
M010: NOP   0;
NETWORK
TITLE = Zielzeiger belegen
//Ziel vom Typ "ANY" erstellen
      LAR1  P##Zielzeiger;
      L     B#16#10;
      T     LB [AR1,P#0.0];	//Syntax-ID ist immer 10h bei AWL
      L     2;
      T     LB [AR1,P#1.0];	// Datentyp = 2 (Byte)
      L     #Block_Laenge;
      T     LW [AR1,P#2.0];	// Anzahl der Bytes die kopiert werden sollen
      L     #Ziel_DB;
      T     LW [AR1,P#4.0];	// Datenbaustzeinnummer
      L     #Operandenbereich;
      L     128;	// 128 addieren (Bit 31 muß 1 sein)
      +I;
      SLD   24;	// 24 Stellen nach rechts schieben
      L     #Ziel_DW;
      SLD   3;	// Quell-DW an Byte-Adresse schieben 
      +D;	// Zeiger zusammenfügen
      T     LD [AR1,P#6.0];	// siehe Aufbau Bereichszeiger NW1
NETWORK
TITLE = Blocktransfer
//Blocktransfer mit Systemfunktion SFC20
      CALL  "BLKMOV" (
           SRCBLK                   := #Quellzeiger,
           RET_VAL                  := #SFC20_return,
           DSTBLK                   := #Zielzeiger);
NETWORK
TITLE = Rückgabewert SFC20
//Rückgabewert des SFC20 übergeben
      L     #SFC20_return;
      T     #outFehler;
END_FUNCTION

FUNCTION "FC6 Datenbit zuw./abfr." : VOID	// FC 6
TITLE = Datenbit_setzen oder abfragen ( Adressierung Byte )
//Erstellung:
//Datum        Bearbeiter                                                 Version
//--------------------------------------------------------------------------------
//26.06.97     H.Rüttling (rh)                                            01.00.00
//
//Änderungen:
//Nr. Datum    Bearb Beschreibung                                   Marke Version
//--------------------------------------------------------------------------------
//01  12.11.98 sra   komplette Überarbeitung                              02.00.00
//02  20.11.98 gea   Vereinfachung                                        02.00.01
//03  24.09.14 sra   Adresserweiterung (>8192)                      (003) 02.01.00
//________________________________________________________________________________
//Funktion:
//
//Die Funktion schreibt oder liest den Zustand eines Datenbits.
//Das Datenbit ist definiert durch Datenbaustein [in_DB_Nr], die 
//Anfangsbytenummer [in_Byte_Nr_Anfang] und die Bitnummer [in_Bit_Nr].
//Ist der Parameter in_Mode_Z_A = 'A' wird das Datenbit gelesen und in den 
//Parameter io_Wert geschrieben.
//Ist der Parameter in_Mode_Z_A = 'Z' wird das Datenbit entsprechende dem Zustand 
//des Parameters io_Wert geschrieben.
//
//Es können auch Bitnummern > 7 verwendet werden. Dann wird die Bytenummer 
//entsprechend dem Vielfachen von 8 erhöht.
//Z.B.: Byte 8, Bit 12 entspricht Byte 9, Bit 4
//
//!!!! in_Bit_Nr.= 0 => DBX Byte X.0 !!!!!
//!!!! in_Bit_Nr.= 1 => DBX Byte X.1 !!!!!
AUTHOR : rh
FAMILY : AZO
VERSION : 0.0
VAR_INPUT
  in_DB_Nr : INT ;	//Datenbausteinnummer
  in_Byte_Nr_Anfang : INT ;	//Byte-Nummer
  in_Bit_Nr : INT ;	//Bitnummer
  in_Mode_Z_A : CHAR ;	//Z = zuweisen; A = abfragen
END_VAR
VAR_IN_OUT
  io_Wert : BOOL ;	//Wert der gelesen/geschrieben wird
END_VAR
VAR_TEMP
  Datenbaustein : INT ;
  Byte_Adresse : INT ;
  Bit_Adresse : INT ;
END_VAR
BEGIN
NETWORK
TITLE = Datenbaustein aufschlagen
      L     #in_DB_Nr;	// Datenbaustein_NR uebergeben
      T     #Datenbaustein;
      OPN   DB [#Datenbaustein];	// Datenbaustein indiziert aufschlagen
NETWORK
TITLE = Byte Adresse berechnen
      L     #in_Bit_Nr;
      SRW   3;	// Bit_ NR durch 8 dividieren
      L     #in_Byte_Nr_Anfang;	// Ergebnis zur Wort-Adresse dazuadieren
      +D;	// (003)
      T     #Byte_Adresse;	// = Datenwort Adresse
NETWORK
TITLE = Bit_Adresse berechnen
      L     #in_Bit_Nr;
      L     W#16#7;
      AW;
      T     #Bit_Adresse;
NETWORK
TITLE = Pointer auf Datenbit berechnen
      L     #Byte_Adresse;	// DW Adresse zurecht ruecken
      SLD   3;	// DW Adresse zum Adressregister  // (003)
      L     #Bit_Adresse;	// Bit Adresse hinzufügen
      OD;	// (003)
      LAR1;	// Pointer Adresse aus Adressregister
NETWORK
TITLE = Mode Auswahl
      L     'Z';
      L     #in_Mode_Z_A;
      ==I;
      JC    ZUWE;	// Sprung Datenbit zuweisen
      L     'A';
      ==I;
      JC    ABFR;	// Sprung Datenbit abfragen
      BEU;
NETWORK
TITLE = Datenbit zuweisen 
ZUWE: A     #io_Wert;
      =     DBX [AR1,P#0.0];
      BEU;
NETWORK
TITLE = Datenbit abfragen
ABFR: A     DBX [AR1,P#0.0];
      =     #io_Wert;
END_FUNCTION

FUNCTION "FC7 Tabelle auslesen" : VOID	// FC 7
TITLE = Tabelle auslesen
//Erstellung:
//Datum        Bearbeiter                                                 Version
//--------------------------------------------------------------------------------
//30.10.98     A.Geiger (gea)                                             01.00.00
//
//Änderungen:
//Nr. Datum    Bearb Beschreibung                                   Marke Version
//--------------------------------------------------------------------------------
//01  10.05.99 sra   Bereichszeigerberechnung korrigiert                  01.00.01
//02  29.08.00 gea   Neue Konzeption(Kopieren über Schleife)              02.00.00
//03  26.10.01 gea   Fehlerbehebung DB überprüfen                   (003) 02.00.01
//04  26.10.01 gea   Fehler bei Anfangsbyte negativ                 (004) 02.00.02
//05  29.02.16 sra   Anpassung für Tabellen > 32767 Byte            (005) 02.00.03
//06  17.06.16 sra   Fehlerbeseitigung Zeigerberechnung             
//                   negative Zeilen sind ebenfalls möglich         (006) 02.00.04
//________________________________________________________________________________
//Funktion:
//
//Beschreibung: Datensatz aus Tabelle auslesen
//
//Aufbau Tabellen-DB:
//      DBB(Offset)    ... DBB(n-1)  1.Zeile
//      DBB(Offset+n)  ... DBB(2n-1) 2.Zeile
//      DBB(Offset+2n) ... DBB(3n-1) 3.Zeile
//      usw.
//
//Die Anzahl der Spalten pro Zeile (n) ist abhängig von der Länge des "Ziels".
//Das "Ziel" muß ein ANY-Zeiger auf Bytes oder eine Stuktur sein.
//Eine Überprüfung auf Existenz und Länge des Tabellen-DBs wird durchgeführt.
//
//Fehlermeldungen:
//-1 = Bereichszeiger Quelle falsch
//-2 = Bereichszeiger Ziel falsch
//-3 = Blocklänge falsch
//-4 = Datenbaustein nicht existent 
//-5 = Datenbaustein Längenfehler
//-6 = Fehler Datentyp in ANY-Zeiger
//-7 = Fehler Anfangsbyte negativ    
//
AUTHOR : gea
FAMILY : gea
VERSION : 0.0
VAR_INPUT
  in_Tabelle_DB : INT ;	//Tabellen-DB-Nr.
  in_Offset_DW : INT ;	//Offset erster Tabelleneintrag in Tabellen-DB
  in_Zeile_lesen : INT ;	//Eintrag in Tabelle, der gelesen werden soll
END_VAR
VAR_OUTPUT
  out_Fehler : INT ;	//-1=Q,-2=Z,-3=Blocklänge,-4=DB n. vorh.,-5=DB zu kurz,-6=Datentyp,-7=Anfangsbyte
END_VAR
VAR_IN_OUT
  io_Ziel : ANY ;	//Zeiger auf Zieldaten Block in den kopiert wird
END_VAR
VAR_TEMP
  G_DB_SAVE : INT ;	//Global-DB-Register
  I_DB_SAVE : INT ;	//Instanz-DB-Register
  Zeiger_Quelle : DWORD ;
  DB_Quelle : INT ;
  Zeiger_Ziel : DWORD ;
  DB_Ziel : INT ;
  Blocklaenge : INT ;
  Datentyp : BYTE ;
  Start_DBB : INT ;
END_VAR
BEGIN
NETWORK
TITLE = DB-Register sichern
      L     DBNO;
      T     #G_DB_SAVE;
      L     DINO;
      T     #I_DB_SAVE;
NETWORK
TITLE = ANY-Zeiger Ziel zerlegen
      L     P##io_Ziel;
      LAR1;
      L     B [AR1,P#1.0];
      T     #Datentyp;
      L     W [AR1,P#2.0];
      T     #Blocklaenge;
      L     W [AR1,P#4.0];
      T     #DB_Ziel;
      L     D [AR1,P#6.0];
      L     DW#16#FFFFFF;	// (006)
      AD;	// (006)
      T     #Zeiger_Ziel;
NETWORK
TITLE = Blocklänge prüfen
      L     #Blocklaenge;
      L     0;
      <=I;
      JC    BLFE;	//Blocklänge Fehler
NETWORK
TITLE = Datentyp prüfen
      L     #Datentyp;
      L     2;	//Datentyp = Byte oder Struct
      ==I;
      JCN   DTFE;
NETWORK
TITLE = Start-DBB des gewählten Eintrags
      L     #in_Zeile_lesen;
      L     1;
      -I;
      L     #Blocklaenge;
      *I;
      L     #in_Offset_DW;
      +I;
      T     #Start_DBB;	//Start des n-ten Eintrags
//      L     #Start_DBB                  //Start des n-ten Eintrags      //(004) // (006)
//      L     0                           //                                (004) // (006)
//      >=I                               //                                (004) // (006)
//      SPBN  DBBN                        //Fehler Anfangsbyte negativ    //(004) // (006)
NETWORK
TITLE = Bereichszeiger Quellzeiger
      L     W#16#84;
      CAD;
      L     #Start_DBB;
      SLD   3;
      +D;
      T     #Zeiger_Quelle;
NETWORK
TITLE = Quell-DB
      L     #in_Tabelle_DB;
      T     #DB_Quelle;
NETWORK
TITLE = DBs aufschlagen
//      L     #DB_Quelle                               //(003)
//      L     0                                        //(003)
//      <>I                                            //(003)
//      SPBN  QNDB                                     //(003)
      OPN   DB [#DB_Quelle];
      L     DBNO;
      L     0;
      <=I;
      JC    DBNX;	//Fehler DB existiert nicht
      L     #Start_DBB;
      L     #Blocklaenge;
      +D;	// (005)
      L     DBLG;
      >D;	// (005)
      JC    DBLF;	//Fehler DB Länge nicht ausreichend
      L     #DB_Ziel;
      L     0;
      <>I;
      JCN   ZNDB;
      OPN   DI [#DB_Ziel];
      L     DINO;
      L     0;
      <=I;
      JC    DBNX;	//Fehler DB existiert nicht
      L     #Zeiger_Ziel;
      SRD   3;	//Anfangsbyte (005)
      L     #Blocklaenge;
      +D;	// (005)
      L     DILG;
      >D;	// (005)
      JC    DBLF;	//Fehler DB Länge nicht ausreichend
      L     #Zeiger_Ziel;
      L     DW#16#FFFFFF;
      AD;
      L     W#16#85;
      CAD;
      +D;
      T     #Zeiger_Ziel;
ZNDB: NOP   0;
NETWORK
TITLE = Bytes kopieren
//geschwindigkeitsopitmiert:
//- Schleifenzäehler bleibt in AKKU1 und AKKU2
//- Kopieren über Worte, letztes Byte (ungerade Bytezahl) separat.
// (network holds code this reader does not know; not shown)
NETWORK
TITLE = Fehlerauswertung
      L     0;	//kein Fehler
      JU    SEFE;	//  setze Fehlerausgang
      L     -1;	//Bereichszeiger Quelle falsch
      JU    SEFE;	//  setze Fehlerausgang
      L     -2;	//Bereichszeiger Ziel falsch
      JU    SEFE;	//  setze Fehlerausgang
BLFE: L     -3;	//Blocklänge falsch
      JU    SEFE;	//  setze Fehlerausgang
DBNX: L     -4;	//Datenbaustein nicht existent 
      JU    SEFE;	//  setze Fehlerausgang
DBLF: L     -5;	//Datenbaustein Längenfehler
      JU    SEFE;	//  setze Fehlerausgang
DTFE: L     -6;	//Fehler Datentyp in ANY-Zeiger
      JU    SEFE;	//  setze Fehlerausgang         (004)
      L     -7;	//Fehler Anfangsbyte negativ    (004)
SEFE: T     #out_Fehler;
NETWORK
TITLE = DB-Register wiederherstellen
      OPN   DB [#G_DB_SAVE];
      OPN   DI [#I_DB_SAVE];
NETWORK
TITLE = BIE-Bit zuweisen
      L     #out_Fehler;
      L     0;
      ==I;
      SAVE;
END_FUNCTION

FUNCTION "FC8 ANY-Zeiger zerlegen" : VOID	// FC 8
TITLE = Ermittlung DB, DW, Laenge Anyzeiger
//Erstellung:
//Datum        Bearbeiter                                                 Version
//--------------------------------------------------------------------------------
//03.03.99     A.Geiger (gea)                                             01.00.00
//
//Änderungen:
//Nr. Datum    Bearb Beschreibung                                   Marke Version
//--------------------------------------------------------------------------------
//01  
//
//________________________________________________________________________________
//Funktion:
//
//Der Baustein ermittelt aus einem ANY-Zeiger:
//  Datenbausteinnummer
//  Datenwortnummer Beginn des Anyzeigers
//  Länge des Bereiches in Byte
//
AUTHOR : gea
FAMILY : AZO
VERSION : 0.0
VAR_INPUT
  in_Zeiger : ANY ;	//ANY-Zeiger
END_VAR
VAR_OUTPUT
  out_DB : INT ;	//Datenbausteinnummer
  out_DW : INT ;	//Anfangs-Datenwortnummer
  out_Laenge : INT ;	//Länge des Bereiches in Byte
END_VAR
BEGIN
NETWORK
TITLE = Ermittlung DB, DW, Laenge Anyzeiger
      L     P##in_Zeiger;
      LAR1;
      L     W [AR1,P#2.0];
      T     #out_Laenge;
      L     W [AR1,P#4.0];
      T     #out_DB;
      L     D [AR1,P#6.0];
      SRD   3;
      T     #out_DW;
END_FUNCTION

FUNCTION "FC10 Analogwert r/w" : VOID	// FC 10
TITLE = Analogwert lesen/schreiben
//Erstellung:
//Datum        Bearbeiter                                                 Version
//--------------------------------------------------------------------------------
//06.08.97     G.Herkert (hkt)                                            01.00.00
//
//Änderungen:
//Nr. Datum    Bearb Beschreibung                                   Marke Version
//--------------------------------------------------------------------------------
//01  21.10.97 rh    Drahtbruchüberwachung ergänzt                        01.01.00
//02  05.12.97 rh    Adressen auf PEW und PAW geändert                    01.01.01
//03  25.11.98 gea   Simulation eingefügt                                 01.02.00
//04  29.03.99 gea   Fehlerbehebung Drahtbruchüberwachung                 01.02.01
//05  30.06.99 sra   Fehlerbehebung Drahtbruchüberwachung                 01.02.02
//06  19.02.00 sra   Unterscheidung Drahtbruchüberwachung                 01.02.03
//07  12.09.01 gea   Eingangsparameter in_E_A_Adresse als INT             01.03.00
//08  16.03.04 sra   nicht in Simulations-DB schreiben wenn Simul aus     01.03.01
//09  17.09.08 sra   Wago-System 750-466 erweitert                  (009) 01.04.00
//________________________________________________________________________________
//Funktion:
//
//Der Baustein liest den Wert eines Analogeinganges ein und normiert diesen. Die 
//Normierung erfolgt anhand der Vorgabe der Eingangsparameter Obergrenze und 
//Untergrenze.
//
//Hinweis:
//- bei Siemens-Baugruppen ist der Wert "MaxDigit" = 27648
//- bei Wago-Baugruppen 740-466 ist der Wert "MaxDigit" = 32760
//
//
AUTHOR : hkt
FAMILY : AZO
VERSION : 0.0
VAR_INPUT
  in_E_A : CHAR  := 'E';	//E = Eingang, A = Ausgang
  in_EA_Adresse : INT ;	//Ein-/Ausgangsadresse des Analogkanals
  in_OberGrenze : REAL ;	//Obergrenze des Ausgabewertes (z.B. Drucktransmitter: 2 bar)
  in_UnterGrenze : REAL ;	//Untergrenze des Ausgabewertes (z.B. Drucktransmitter: 0 bar)
  in_MaxDigit : REAL ;	//Digitwert den die Baugruppe bei der Obergrenze liefert z.B. 27648
  in_MinDigit : REAL ;	//Digitwert den die Baugruppe bei der Untergrenze liefert z.B. 0 bzw. -27648
  in_Typ : CHAR ;	//Z=Zentralbaugruppe, B=ET200B Analogmodul, W=Wago 750-466, sonstige
  in_Simulation : BOOL ;	//Simulation des Analogwertes über Eintrag in Datenbaustein
  in_DB_Simulation_EA : INT ;	//Simulation-DB des Analogwertes über Eintrag in Datenbaustein
END_VAR
VAR_IN_OUT
  io_Wert : REAL ;	//eingelesener und normierter Wert den die Baugrppe liefert
  io_Drahtbruch : BOOL ;	//Drahtbruchstoerung
END_VAR
VAR_TEMP
  MaxDigit_MinDigit : REAL ;
  E_MinDigit : REAL ;
  OG_UG : REAL ;
  Eingang_Real : REAL ;
  Pointer_EA_Adresse : DWORD ;
  Wert_analog : WORD ;
  DB_Sim : INT ;
END_VAR
BEGIN
NETWORK
TITLE = Zwischenwerte berechnen
      L     #in_MaxDigit;
      L     #in_MinDigit;
      -R;
      T     #MaxDigit_MinDigit;
      L     #in_OberGrenze;
      L     #in_UnterGrenze;
      -R;
      T     #OG_UG;
NETWORK
TITLE = Zeiger berechnen
// Zeiger auf EA-Adresse berechnen
      LAR1  P#0.0;
      L     #in_EA_Adresse;
      SLW   3;
      +AR1;
      LAR1;
      T     #Pointer_EA_Adresse;	//Zeiger auf EA-Adresse
      L     #in_DB_Simulation_EA;
      T     #DB_Sim;	//Zeiger auf EA-DB
NETWORK
TITLE = Analogwert einlesen
//Analogwert einlesen
//Formel:   Wert = UG + (OG-UG)*(E-MinDigit) / (MaxDigit-MminDigit)
      L     #in_E_A;
      L     'E';
      <>I;
      JC    NotE;
      A     #in_Simulation;
      JC    SIME;
      L     PIW [#Pointer_EA_Adresse];
      JU    WERE;	// (008)
SIME: OPN   DB [#DB_Sim];
      L     DBW [#Pointer_EA_Adresse];
WERE: T     #Wert_analog;
      A(;
      L     #in_Typ;	// Abfrage Drahtbruchüberwachung
      L     'Z';	// "Z" = Zentralbaugruppe
      ==I;
      );
      A(;
      L     #Wert_analog;	// 7FFF Ersatzwert für Drahtbruch
      L     W#16#7FFF;
      ==I;
      );
      O;
      A(;
      L     #in_Typ;	// Abfrage Drahtbruchüberwachung
      L     'B';	// "B" = ET200B Baugruppe
      ==I;
      );
      A(;
      L     #Wert_analog;	// 8000 Ersatzwert für Drahtbruch
      L     W#16#8000;
      ==I;
      );
      O;	// -> (009)
      A(;
      L     #in_Typ;	// Abfrage Kartentyp
      L     'W';	// "W" = Wago System 750-466
      ==I;	// Karte meldet mit den rechten 3 Bis ein Kurzschluss bzw. Überlauf
      );
      A(;
      L     #Wert_analog;
      L     W#16#7;
      AW;
      L     W#16#0;
      <>I;
      );	// <- (009)
      =     #io_Drahtbruch;
      L     #Wert_analog;
      ITD;
      DTR;
      T     #Eingang_Real;
      L     #Eingang_Real;
      L     #in_MinDigit;
      -R;
      T     #E_MinDigit;
      L     #OG_UG;
      L     #E_MinDigit;
      *R;
      L     #MaxDigit_MinDigit;
      /R;
      L     #in_UnterGrenze;
      +R;
      T     #io_Wert;
NotE: NOP   0;
NETWORK
TITLE = AnalogWert ausgeben:  
//AnalogWert ausgeben:
//Formel : A = MinDigit+(MaxDigit-MinDigit)*(Wert-UG)/ (Og-UG)
      L     #in_E_A;
      L     'A';
      <>I;
      JC    NotA;
      L     #io_Wert;
      L     #in_UnterGrenze;
      -R;
      L     #OG_UG;
      /R;
      L     #MaxDigit_MinDigit;
      *R;
      L     #in_MinDigit;
      +R;
      RND;
      T     #Wert_analog;
      A     #in_Simulation;
      JC    SIMA;
      T     PQW [#Pointer_EA_Adresse];
      JU    NotA;	// (008)
SIMA: OPN   DB [#DB_Sim];
      T     DBW [#Pointer_EA_Adresse];
NotA: NOP   0;
END_FUNCTION

FUNCTION "FC13 Standardsignale" : VOID	// FC 13
TITLE = Baustein für Standardmerker
//Erstellung:
//Datum        Bearbeiter                                                 Version
//--------------------------------------------------------------------------------
//26.06.97     R.Schaffert (sra)                                          01.00.00
//
//Änderungen:
//Nr. Datum    Bearb Änderung                                       Marke  Version
//--------------------------------------------------------------------------------
//01  21.11.02 sra   Resetmerker eingefügt                          (001) 01.00.01
//02  30.08.12 pti   Lampe Steuerspannung ein eingefügt             (002) 01.01.00
//03  23.07.13 sra   Signale für Sicherung eingefügt                (003) 01.02.00
//04  05.12.13 sra   Signal Steuerspannung gelöscht                       01.03.00
//05  02.06.14 sra   M0.3 Reset ebenfalls gelöscht (zu Änderung 04)       01.03.01
//06  14.12.16 sra   Implement SFC51 to read battery information    (006) 01.04.00
//________________________________________________________________________________
//Funktion:
//  
//Der Baustein erzeugt folgende Standardsignale:
//- M 0.1 "konstant 1" Merker
//- M 0.2 "konstant 0" Merker
//- M 1.6 Melderentprelltakt (5 Sekunden) 
//- M 1.7 "Takt Timernachbildung" = in_Basistakt_Timer
//- MB4 Impulsmerker für Takte 2.0s, 1.6s, 1.0s, 0.8s, 0.5s, 0.4s, 0.2s, 0.1s
//  !!! MB 2 muss als Taktmerker in CPU parametriert werden  !!
//  Das MB 3 wird als Hilfsbyte zur Flankenauswertung benutzt
//- MW 6 Zeitwert Takt = in_Zeit_Basistakt_100ms
AUTHOR : sra
FAMILY : AZO
VERSION : 0.0
VAR_INPUT
  in_E_Sicherung_OK : BOOL ;	//Eingang Sicherung OK = Eingang Störung Sicherung
  in_Basistakt_Timer : BOOL ;	//Taktmerker für alle Zeitfunktionen (abhängig von Zykluszeit)
  in_Zeit_Basistakt_100ms : INT ;	//Zeitwert Basistakt in 100 ms
END_VAR
VAR_OUTPUT
  o_Lampe_Stoer_Sicherung : BOOL ;	//Ausgang der Lampe "Störung Sicherung"
  o_Stoerung_Sicherung : BOOL ;	//Störung Sicherung -> für Störbitzuweisung im DB34
END_VAR
VAR_TEMP
  NOP : INT ;
END_VAR
BEGIN
NETWORK
TITLE = Statische Merker  
      SET;
      S     "M0.1 Constant1";
      R     "M0.2 Constant0";
NETWORK
TITLE = Lampe "Störung Sicherung" und Störmeldung Sicherung
//(003)
      AN    #in_E_Sicherung_OK;
      =     #o_Lampe_Stoer_Sicherung;
      =     #o_Stoerung_Sicherung;
NETWORK
TITLE = Impulsmerker Takte
//Impulsmerker für Takte 2.0s, 1.6s, 1.0s, 0.8s, 0.5s, 0.4s, 0.2s, 0.1s
//positive Flankenauswertung auf die von der CPU erzeugten Takte
      L     MB 3;
      L     MB 2;
      T     MB 3;
      XOW;
      L     MB 2;
      AW;
      T     MB 4;
NETWORK
TITLE = Werte für Timernachbildung vorgeben
//!! Abhängig von Zykluszeit !! 
      A     #in_Basistakt_Timer;
      =     "M1.7 ClockTimerFunction";
      L     #in_Zeit_Basistakt_100ms;
      T     "MW 6 Timer Val Cycle FCs";
NETWORK
TITLE = Takt Melderentprellung
//Takt Melderentprellung
      AN    "M1.6 ClockLevelIndicato";
      L     S5T#5S;
      SD    T 1;
      A     T 1;
      =     "M1.6 ClockLevelIndicato";
NETWORK
TITLE = read Battery fault of CPU
//(006)
      CALL  "RDSYSST" (
           REQ                      := "M2.7 Flag2,0Sec",
           SZL_ID                   := W#16#392,
           INDEX                    := W#16#0,
           RET_VAL                  := "DB3 CPU Daten".RDSYSST.RETVAL,
           BUSY                     := "DB3 CPU Daten".RDSYSST.BUSY,
           SZL_HEADER               := "DB3 CPU Daten".RDSYSST.SLZ_HEADER,
           DR                       := "DB3 CPU Daten".RDSYSST.DR);	// W#16#392 = Status of the backup batteries in a rack/module rack of a CPU after at least one battery has failed /  if ID = 392h -> Index is always 0
      L     "DB3 CPU Daten".RDSYSST.DR.Data_1;
      L     0;
      <>I;
      =     "DB3 CPU Daten".Fehler_OB_Info.Battery_fault;
END_FUNCTION

FUNCTION "FC16 Störauswertung" : VOID	// FC 16
TITLE = Sammelstoerung
//Erstellung:
//Datum        Bearbeiter                                                 Version
//--------------------------------------------------------------------------------
//26.07.99     M.Junker (jm)                                              01.00.00
//
//Änderungen:
//Nr. Datum    Bearb Änderung                                       Marke  Version
//--------------------------------------------------------------------------------
//01  14.09.99 jm    Spiegelung von PC ergänzt                            01.01.00
//02  06.10.99 jm    Störauswertung DWORD-weise                           01.02.00
//03  23.10.99 jm    QuitierungsDWORD von PC löschen                      01.03.00
//04  03.11.99 jm    Fehlerbeseitigung: QIP und DWORD                     01.03.01
//05  27.03.00 jm    Fehlerbeseitigung DWORD (Erstmeldung)                01.03.02
//06  19.04.05 jm    Fehlerbeseitigung Pointeradressen >8192(=>SLD) (006) 01.03.03
//07  23.02.06 jm    Quittierungs-DB Farbgrafik ist extern
//                   => Quittierung üder Kastor oder Farbgrafik     (007) 01.04.00
//08  23.03.06 sra   Einzelstörungsbereiche
//                   +Quitt.Erstwertmeldung über Quittierbereich         
//                   +Erstwertmeldung löschen ohne Störung          (008) 01.05.00
//09  10.05.06 sra   Fehlerbeseitigung zu Änderung 08               (009) 01.05.01
//10  11.05.06 sra   Änderung Quittierung von Farbgrafik            (010) 01.05.02
//11  05.10.06 jm    Anpassung für Siemens OP: extra Quittierbereich
//                   mit Flankenauswertung                          (011) 01.06.00
//12  01.04.08 jm    Steuerspannung entfernt, da Probleme mit OP-
//                   Quittierung (Problem: vorhandene Störung bei
//                   Steuerspannung aus am OP quittieren)           (012) 01.06.01
//13  16.11.15 sra   "Steuerspannung" in "Frg. Sammenstörung" geänd.(013) 01.06.02
//________________________________________________________________________________
//Beschreibung:
//
//!!!ACHTUNG: Parameter Anzahl Störungsbyte muß immer durch 4 teilbar sein!!!!
//
//Der Baustein überwacht einen definierbaren Teil eines Datenbaustein (DB34) in 
//dem alle Störmeldungen gesammelt werden. Sobald eine Störung vorhanden ist wird 
//das Signal "Sammelstörung" gebildet um damit z.B. eine Sammelstörlampe 
//anzusteuern. Der Parameter "Anzahl Störungsbyte" muß immer durch 4 teilbar sein
//
//In weiteren Bereichen weden die Datenblöcke "Erstmeldung", "Erstmeldung PC" und 
//Quittierung PC" mit der gleichen Größe wie der Störbereich benötigt.
//
//Funktion:
//Um bei der Störungsquittierung zur FG kompatibel zu sein werden die 
//Quittierungen, sobald die Störung verschwunden ist, von der SPS gelöscht.
//
//Die beiden Quittierungsbereiche (in DB34 für Kastor; in DB35 für SCADA) werden 
//mit ODER ausgewertet, d.h. die Störungen könnten von beiden Seiten quittiert 
//werden (wird normal nicht gemacht). Die Quittierbits werden hier so umkopiert, 
//daß sie immer in beiden Quittierungsbereichen auftauchen.
//=> es müssen immer beide Quittierbereiche angelegt sein
//=> an den Aggregat-Baustein werden die Bits aus dem DB35 angelegt
//
//OP:
//Siemens OPs müssen in einen extra Bereich quittieren, der hinter dem normalen 
//Standardbereichen im DB34 liegt. Im Anschluss folgt noch ein Bereich für die 
//Flankenauswertung. Bei positiver Flanke der Quittierung von OP wird die in den 
//Bereich der SCADA-Quittierung übertragen. In den OP Quittierbereich darf auf 
//gar keinen Fall die SPS schreiben. Wird kein OP verwendet so können die 
//OP-Bereiche aus dem DB34 weggelassen werden.
AUTHOR : jm
FAMILY : STANDARD
NAME : hsh
VERSION : 0.0
VAR_INPUT
  Conf_AckBySiemensOP : BOOL ;	//configuration bit: ackowledge done by Siemens OP (011)
  Stoerungstakt : BOOL ;	//Takt für Störauswertung
  Freigabe_Sammelstoerung : BOOL ;	//Freigabe Sammelstörung (ehemals Steuerspannung)
  Quittierung : BOOL ;	//Quittierung Fehlermeldung
  Stoerungs_DB : INT ;	//Stör-Datenbaustein
  Quittierungs_DB_SCADA : INT ;	//Quittier-Datenbaustein Farbgrafik
  Anzahl_Stoerungs_Byte : INT ;	//Anzahl Störungsbyte im Stör-Db (Blocklänge der 4 Bereiche)
  Offset_Stoerungs_Byte : INT ;	//Anfangs-DW der Störmeldungen im Stör-DB (wenn Bereich nicht bei Byte 0 anfängt)
  Adresse_Anfangswort : INT ;	//Adresse des ersten Datenwortes das ausgewertet wird
  Bereichslaenge : INT ;	//Länge des Bereiches der ausgewertet wird (!!Muss durch 4 teilbar sein!!)
END_VAR
VAR_IN_OUT
  Sammelstoerung : BOOL ;	//Sammelstörung
  Erstmeldung : BOOL ;	//Erstmeldung aktiv
  Erstmeldung_PC : BOOL ;	//Erstmeldung an PC
  Quittierung_PC : BOOL ;	//Quittierung von PC
END_VAR
VAR_TEMP
  Stoer_DB : INT ;	//Stoerungs-DB lokal
  Quit_DB : INT ;	//Quittierungs-DB extern
  Offsetende : INT ;	//= Störungsbyte + Offset
  SI : INT ;	//Störungsindex
  KI : INT ;	//Kopierindex
  SIP : INT ;	//Spiegelungsindex PC
  QIP : INT ;	//Quittierungsindex PC
  QIS : INT ;	//Quitierungsindex SCADA
  QIO : INT ;	//Quittierungsindex Siemens OP (011)
  KQIO : INT ;	//Kopie Quittierungsindex Siemens OP (011)
  StoerungsDWORD : DWORD ;	//Stoerungsdoppelwort
  KopieDWORD : DWORD ;	//Kopiedoppelwort
  SpiegelungsDWORD : DWORD ;	//Spiegelungsdoppelwort
  QuittierungsDWORD : DWORD ;	//Quittierungsdoppelwort
  QuitPC_DWORD : DWORD ;	//Quittierungsdoppelwort von PC
  QuitSCADA_DWORD : DWORD ;	//Quittierungsdoppelwort von SCADA
  QuitOP_DWORD : DWORD ;	//Quittierungdoppelwort von OP (011)
  KopieQuitOP_DWORD : DWORD ;	//Kopie Quittierungdoppelwort von OP (011)
  t_Erstmeldung_PC : BOOL ;	//Erstmeldung an PC
END_VAR
BEGIN
NETWORK
TITLE = Störauswertung aktiv?
//      ON    #Steuerspannung // (012)
//      SPB   FCEN                       // FunCtion ENd // (012)
      ON    #Stoerungstakt;
      JC    QUIT;	// QUITtierung Erstmeldung prüfen
NETWORK
TITLE = Variablen vorbelegen
//Minus 4 wegen DWORD-Auswertung
      CLR;
      =     #Sammelstoerung;
      =     #t_Erstmeldung_PC;
      L     #Offset_Stoerungs_Byte;
      L     #Adresse_Anfangswort;	// (008)
      +I;	// (008)
      L     #Bereichslaenge;	// (008)
      +I;
      T     #Offsetende;	//Offsetende = Offset + Anzahl // (007)
      L     #Offsetende;	// (007)
      L     4;
      -I;
      T     #SI;	//Stoerungsindex = Offsetende + Anzahl -4
      T     #QIS;	//Quittierungsindex SCADA = Stoerungsindex (007)
      L     #Offsetende;	// (007)
      L     #Anzahl_Stoerungs_Byte;	// (008)
      +I;
      L     4;
      -I;
      T     #KI;	//Kopierindex = Offsetende + Anzahl*2 -4
      L     #Offsetende;	// (007)
      L     #Anzahl_Stoerungs_Byte;
      +I;
      L     #Anzahl_Stoerungs_Byte;	// (008)
      +I;
      L     4;
      -I;
      T     #SIP;	//Spiegelungsindex PC = Offsetende + Anzahl*3 -4
      L     #Offsetende;	// (007)
      L     #Anzahl_Stoerungs_Byte;
      +I;
      L     #Anzahl_Stoerungs_Byte;
      +I;
      L     #Anzahl_Stoerungs_Byte;	// (008)
      +I;
      L     4;
      -I;
      T     #QIP;	//Quittierungsindex PC = Offsetende + Anzahl*4 -4
// >>>>>>>>>> (011)
      L     #Offsetende;
      L     #Anzahl_Stoerungs_Byte;
      +I;
      L     #Anzahl_Stoerungs_Byte;
      +I;
      L     #Anzahl_Stoerungs_Byte;
      +I;
      L     #Anzahl_Stoerungs_Byte;
      +I;
      L     4;
      -I;
      T     #QIO;	//Quittierungsindex OP = Offsetende + Anzahl*5 -4
      L     #Offsetende;
      L     #Anzahl_Stoerungs_Byte;
      +I;
      L     #Anzahl_Stoerungs_Byte;
      +I;
      L     #Anzahl_Stoerungs_Byte;
      +I;
      L     #Anzahl_Stoerungs_Byte;
      +I;
      L     #Anzahl_Stoerungs_Byte;
      +I;
      L     4;
      -I;
      T     #KQIO;	//Kopie Quittierungsindex OP = Offsetende + Anzahl*6 -4
// <<<<<<<<<< (011)
NETWORK
TITLE = Störungs-/Kopie-/Spiegelungs-/QuittierungsDWORD(OP) laden
      L     #Stoerungs_DB;
      T     #Stoer_DB;
      L     #Quittierungs_DB_SCADA;	// (007)
      T     #Quit_DB;	// (007)
SLOP: OPN   DB [#Stoer_DB];
      L     #SI;
      SLD   3;	// (006)
      LAR1;
      L     DBD [AR1,P#0.0];
      T     #StoerungsDWORD;
      L     #KI;
      SLD   3;	// (006)
      LAR1;
      L     DBD [AR1,P#0.0];
      T     #KopieDWORD;
      L     #SIP;
      SLD   3;	// (006)
      LAR1;
      L     DBD [AR1,P#0.0];
      T     #SpiegelungsDWORD;
      L     #QIP;
      SLD   3;	// (006)
      LAR1;
      L     DBD [AR1,P#0.0];
      T     #QuitPC_DWORD;	// (007)
///*(007)
      L     L#0;	// (011)
      T     #QuitSCADA_DWORD;
      L     #Quittierungs_DB_SCADA;	// (011)
      L     0;
      ==I;	// (011)
      JC    KQ1;	// (011) kein Quittierungsbaustein vorhanden
      OPN   DB [#Quit_DB];
      L     #QIS;
      SLD   3;
      LAR1;
      L     DBD [AR1,P#0.0];
      T     #QuitSCADA_DWORD;
      OPN   DB [#Stoer_DB];
//(007)*/
// >>>>>>>>>> (011)
      L     0;
      T     #QuitOP_DWORD;	// vorbelegen, falls nicht vorhanden
      AN    #Conf_AckBySiemensOP;
      JC    NOPA;	// No OP Acknowledge
      L     #QIO;
      SLD   3;
      LAR1;
      L     DBD [AR1,P#0.0];
      T     #QuitOP_DWORD;
      L     #KQIO;
      SLD   3;
      LAR1;
      L     DBD [AR1,P#0.0];
      T     #KopieQuitOP_DWORD;
NOPA: NOP   0;	// No OP Acknowledge
// <<<<<<<<<< (011)
KQ1:  NOP   0;
NETWORK
TITLE = Pos.Flanke Quittierung OP
//(011)
      AN    #Conf_AckBySiemensOP;
      JC    NPOA;	// No Processing of Op Acknowledge
      L     #QuitOP_DWORD;	// -
      L     #KopieQuitOP_DWORD;	// |
      XOD;	// | positive Flanke Quittierung OP
      L     #QuitOP_DWORD;	// |
      AD;	// -
      L     #QuitSCADA_DWORD;
      OD;
      T     #QuitSCADA_DWORD;	// => Quittierung in QuitSCADA setzen
      L     #QuitOP_DWORD;
      T     #KopieQuitOP_DWORD;	// => Hilfsmerker Flanke (Kopie ALT)
NETWORK
TITLE = Quittierung OP DWORD nach Kopiebyte
//(011)
      L     #KQIO;
      SLD   3;
      LAR1;
      L     #KopieQuitOP_DWORD;
      T     DBD [AR1,P#0.0];	// => Quittierung OP merken
NPOA: NOP   0;
NETWORK
TITLE = Sammelstörung
      L     #StoerungsDWORD;
      L     0;
      <>D;
      A     #Freigabe_Sammelstoerung;	// (012)
      S     #Sammelstoerung;
NETWORK
TITLE = Erstwertmeldung
      L     #StoerungsDWORD;
      L     #KopieDWORD;
      XOD;
      L     #StoerungsDWORD;
      AD;
      L     0;
      <>D;
      A     #Freigabe_Sammelstoerung;	// (012)
      S     #Erstmeldung;
NETWORK
TITLE = Erstwertmeldung an PC
      L     #StoerungsDWORD;
      L     #SpiegelungsDWORD;
      <>D;
      S     #t_Erstmeldung_PC;
NETWORK
TITLE = StoerungsDWORD nach Kopiebyte
      L     #KI;
      SLD   3;	// (006)
      LAR1;
      L     #StoerungsDWORD;
      T     DBD [AR1,P#0.0];
NETWORK
TITLE = neue Quittierung?
//(008)
      L     #QuitSCADA_DWORD;
      L     #QuitPC_DWORD;
      XOD;
      L     0;
      <>D;
      R     #Erstmeldung;
NETWORK
TITLE = QuittierungsDWORD bilden
//(007)
      L     #QuitPC_DWORD;	// (010)
      L     #SpiegelungsDWORD;	// (010)
      AD;	// (010)
      L     #QuitSCADA_DWORD;
      OD;
      T     #QuittierungsDWORD;	// Quittierung von Kastor oder SCADA
NETWORK
TITLE = QuittierungsDWORD löschen
      L     #StoerungsDWORD;
      L     #QuittierungsDWORD;
      AD;
      T     #QuittierungsDWORD;
NETWORK
TITLE = QuittierungsDWORD PC und SCADA löschen
      L     #QIP;
      SLD   3;	// (006)
      LAR1;
      L     #QuittierungsDWORD;
      T     DBD [AR1,P#0.0];	// PC Quittierung
      L     #Quittierungs_DB_SCADA;	// (011)
      L     0;	// (011)
      ==I;	// (011)
      JC    KQ2;	// (011) kein Quittierungsbaustein vorhanden
///*(007)
      OPN   DB [#Quit_DB];
      L     #QIS;
      SLD   3;
      LAR1;
      L     #QuittierungsDWORD;
      T     DBD [AR1,P#0.0];	// SCADA Quittierung
//(007)*/
KQ2:  NOP   0;
NETWORK
TITLE = Störungsschleife von (Anzahl - 4) bis 0
//Minus 4 wegen DWORD-Auswertung
// >>>>>>>>>> (011)
      L     #KQIO;
      L     4;
      -I;
      T     #KQIO;
      L     #QIO;
      L     4;
      -I;
      T     #QIO;
// <<<<<<<<<< (011)
///*(007)
      L     #QIS;
      L     4;
      -I;
      T     #QIS;
//(007)*/
      L     #QIP;
      L     4;
      -I;
      T     #QIP;
      L     #SIP;
      L     4;
      -I;
      T     #SIP;
      L     #KI;
      L     4;
      -I;
      T     #KI;
      L     #SI;
      L     4;
      -I;
      T     #SI;
      L     #Offset_Stoerungs_Byte;
      L     #Adresse_Anfangswort;	// (008)
      +I;	// (008)
      L     #SI;	// (008)
      <=I;	// (008) (009)
      JC    SLOP;	// Störungs LOOP
NETWORK
TITLE = Störauswertung für PC aktiv?
      O     #Erstmeldung_PC;
      O     #Quittierung_PC;
      JC    QUIT;	//QUITtierung
      A     #t_Erstmeldung_PC;
      S     #Erstmeldung_PC;
NETWORK
TITLE = Erstmeldung quittiert?
QUIT: A     #Quittierung;	//QUITtierung
      ON    #Sammelstoerung;	// (008)
      R     #Erstmeldung;
      A     #Quittierung_PC;
      R     #Erstmeldung_PC;
      NOP   0;
END_FUNCTION

FUNCTION "FC20 Motor 1A1E" : VOID	// FC 20
TITLE = Block for motor actuation and fault monitoring
//Erstellung:
//Datum        Bearbeiter                                                 Version
//--------------------------------------------------------------------------------
//26.06.97     H.Rüttling (rh)                                            01.00.00
//
//Änderungen:
//Nr. Datum    Bearb Änderung                                       Marke  Version
//--------------------------------------------------------------------------------
//01  09.02.99 sra   Einfügen der Handbedienuung                    ()    01.01.00
//02  16.04.99 sra   Fehlerbeseitigung Störungsquittierung          ()    01.01.01
//03  23.07.99 sra   Ausg. wird auch bei Simulation gesetzt         ()    01.01.02
//04  19.10.99 sra   "in" Reparaturschalter gelöscht                ()    01.02.00
//05  03.11.99 hus   Parameter eingefügt "FU in Betrieb"            ()    01.03.00
//06  18.09.00 sra   komplette Überarbeitung / neue Struktur        ()    02.00.00
//07  08.11.02 sra   Änderung Betriebsstundenzähler (zählt falsch)  (007) 02.01.00
//08  31.10.05 sra   Ansteuerung Handbedienung im Automode rücksetz.
//                   Handbedienung zentral sperren                  (008) 02.02.00
//09  04.09.06 sra   Änderung Störungsquittierung                   (009) 02.03.00
//10  20.11.07 gea   Handmode zurücksetzen wenn Handmode gesperrt   (010) 02.03.01
//11  18.02.09 kmj   Objektststatus für OP ergänzt                  (011) 02.04.00
//12  20.03.09 kal   Objektststatus für OP ergänzt (überarbeitet)   (012) 02.04.01
//13  05.12.13 sra   "Anlage ein" eingefügt (Not-Aus-Konzept)       (013) 02.05.00
//________________________________________________________________________________
//Funktion:
//
//-Der Baustein steuert den Ablauf eines Motors mit 1 Ausgang und 1 Eingang durch 
// setzten des Eingangsparameters "in_Ansteuerung_Motor".
//
//-Der Ausgang wird nur angesteuert wenn der Eingang "in_Anlage_ein" = true
// ist. Diese Funktion ist vorhanden, um bei einem Not-Halt die Anlage vor 
// unkontrolliertem Einschalten zu schützen. 
//
//-Ist in der Motorstruktur die Taktfunktion freigegeben wird bei Freigabe des 
// Motors der Ausgang entsprechend der Impuls-/Pausezeit angesteuert.
// !!Der Baustein arbeitet nur mit vollen Sekunden!!
//
//-Der Baustein überwacht den Zustand des Ausgangs und des Eingangs und generiert 
// nach Ablauf der "Sollzeit Störung" eine Störmeldung
//
//-Ist das Bit "Simulation" auf TRUE, so wird der Eingang simuliert.
//
//-Ist die Kennung "Betriebsstundenzähler_ein" aktiviert werden die Laufzeit 
// des Motors aufsummiert. Dies erfolgt mit setzen des Ausgangs.
//
//-Der Baustein kopiert die Parameter "in_Eingang_Motor", "io_Ausgang_Motor", 
// "in_Quitt_Stoerung" und "io_Stoerung" in die angegebene Datenstruktur zur 
// Visualisierung auf einem Farbgrafiksystem. Diese Parameter müssen folglich 
// nicht mehr extern umkopiert werden.
//
//-Ist der Parameter "in_Handbedienung_erlaubt" angewählt kann der Motor über 
// eine Farbgrafik oder ein Bedienterminal manuell angesteuert werden
//
AUTHOR : rh
FAMILY : AZO
VERSION : 0.0
VAR_INPUT
  in_Handbedienung_erlaubt : BOOL ;	//1 = manual operation permitted, 0 = manual operation not permitted/locked
  in_Quitt_Stoerung_noetig : BOOL ;	//1 = fault acknowledgement required, 0 = automatic fault acknowledgement
  in_Anlage_ein : BOOL ;	//Anlage bzw. Anlagenbereich nach Not-Halt freigegeben
  in_Quitt_Stoerung : BOOL ;	//Fault acknowledgement when fault_acknowledgement_required = 1
  in_Ansteuerung_Motor : BOOL ;	//Actuation of motor in automatic mode
  in_Eingang_Motor : BOOL ;	//Input of motor
END_VAR
VAR_IN_OUT
  io_Ausgang_Motor : BOOL ;	//Output of motor
  io_Motor_in_Betrieb : BOOL ;	//Signal "motor in operation"
  io_Stoerung : BOOL ;	//Signal "motor fault"
  io_Motorstruktur : ANY ;	//ANY pointer of motor structure
END_VAR
VAR_TEMP
  Freigabe_Takt : BOOL ;
  Start_mit_Impuls : BOOL ;
  Dauertakt : BOOL ;
  Taktausgang : BOOL ;
  Taktanzahl_erreicht : BOOL ;
  Diskrepanz : BOOL ;
  Impulszeit : REAL ;
  Pausezeit : REAL ;
  Sollanzahl_Takte : INT ;
  Zeitzaehler : REAL ;
  Taktzaehler : INT ;
  Objektstatus : INT ;
END_VAR
BEGIN
NETWORK
TITLE = Anfangs-DW der Struktur aus ANY-Zeiger auslesen
      L     P##io_Motorstruktur;
      LAR2;
      L     D [AR2,P#6.0];
      LAR2;
NETWORK
TITLE = Simulation
      AN    DIX [AR2,P#3.5];	// Simulation ein (Struktur)
      JC    ESIM;
      A     #io_Ausgang_Motor;
      =     #in_Eingang_Motor;
ESIM: NOP   0;
NETWORK
TITLE = Umschaltung Hand-/Automatikmode 
      A     DIX [AR2,P#2.7];	// Handmode von Farbgrafik (Struktur)
      AN    DIX [AR2,P#3.1];	// Handmode gesperrt (Struktur)
      AN    "M0.0 LockManualMode";	// Handbedienung zentral sperren (008)
      S     DIX [AR2,P#2.6];	// Handmode zu Farbgrafik (Struktur)
      ON    DIX [AR2,P#2.7];	// Handmode von Farbgrafik (Struktur)
      ON    #in_Handbedienung_erlaubt;
      O     "M0.0 LockManualMode";	// Handbedienung zentral sperren (008)
      O     DIX [AR2,P#3.1];	// Handmode gesperrt (Struktur)//(010)
      R     DIX [AR2,P#2.6];	// Handmode zu Farbgrafik (Struktur)
      R     DIX [AR2,P#2.7];	// Handmode zu Farbgrafik (Struktur) (008)
NETWORK
TITLE = Ansteuerung Handmode zurücksetzen
//(008) 
      AN    DIX [AR2,P#2.6];	// Handmode zu Farbgrafik (Struktur)
      R     DIX [AR2,P#3.0];	// Ansteuerung Handmode von Farbgrafik (Struktur)
NETWORK
TITLE = Daten für Takt in temporäre Variablen laden
      A     #in_Anlage_ein;	// (013)
      A     #in_Ansteuerung_Motor;
      A     DIX [AR2,P#3.6];	// Freigabe Takt (Struktur)
      =     #Freigabe_Takt;
      A     DIX [AR2,P#3.2];	// Start mit Impuls (Struktur)
      =     #Start_mit_Impuls;
      A     DIX [AR2,P#3.3];	// Taktanzahl erreicht (Struktur)
      =     #Taktanzahl_erreicht;
      A     DIX [AR2,P#3.4];	// Dauertakt (Struktur)
      =     #Dauertakt;
      A     DIX [AR2,P#3.7];	// Taktausgang (Struktur)
      =     #Taktausgang;
      L     DID [AR2,P#8.0];	// Impulszeit (Struktur)
      T     #Impulszeit;
      L     DID [AR2,P#12.0];	// Pausezeit (Struktur)
      T     #Pausezeit;
      L     DIW [AR2,P#20.0];	// Sollanzahl Takte (Struktur)
      T     #Sollanzahl_Takte;
      L     DID [AR2,P#16.0];	// Impuls-/Pausezähler (Struktur)
      T     #Zeitzaehler;
      L     DIW [AR2,P#22.0];	// Taktzähler (Struktur)
      T     #Taktzaehler;
NETWORK
TITLE = Takt generieren
      CALL  "FC2 Taktgeber_Timernachb" (
           in_Freigabe              := #Freigabe_Takt,
           in_Rueckmeldung          := #in_Eingang_Motor,
           in_Start_mit_Impuls      := #Start_mit_Impuls,
           in_Dauertakt             := #Dauertakt,
           in_Impuls                := "M4.5 ImpulseClock1,0Sec",
           in_Impulszeit_in_100ms   := 10,
           in_Impulszeit            := #Impulszeit,
           in_Pausezeit             := #Pausezeit,
           in_Sollanzahl_Takte      := #Sollanzahl_Takte,
           io_Taktausgang           := #Taktausgang,
           io_Taktanzahl_erreicht   := #Taktanzahl_erreicht,
           io_Zeitzaehler           := #Zeitzaehler,
           io_Taktzaehler           := #Taktzaehler);
NETWORK
TITLE = Ansteuerung Ausgang des Motors
      A     #in_Anlage_ein;	// (013)
      AN    DIX [AR2,P#2.2];	// Motor gesperrt (Struktur)
      A(;
      AN    #in_Quitt_Stoerung_noetig;
      O;
      A     #in_Quitt_Stoerung_noetig;	// Wenn die Stoerung quittiert werden muß 
      AN    #io_Stoerung;	// wird der Ausgang bei einer anstehenden
      );	// Stoerung zurück gesetzt
      A(;
      AN    DIX [AR2,P#2.6];	// Automatikmode zu Farbgrafik (Struktur)
      AN    DIX [AR2,P#3.6];	// Freigabe Takt (Struktur)
      A     #in_Ansteuerung_Motor;
      O;
      AN    DIX [AR2,P#2.6];	// Automatikmode zu Farbgrafik (Struktur)
      A     DIX [AR2,P#3.6];	// Freigabe Takt (Struktur)
      A     #Taktausgang;
      O;
      A     DIX [AR2,P#2.6];	// Handmode zu Farbgrafik (Struktur)
      A     DIX [AR2,P#3.0];	// Ansteuerung Handmode von Farbgrafik (Struktur)
      );
      O;
      A     #in_Anlage_ein;	// (013)
      A     DIX [AR2,P#24.0];	// FU in Betrieb (Struktur)              
      A     #io_Ausgang_Motor;	// Ausschalten nur möglich, wenn Bit = 0 
      =     #io_Ausgang_Motor;
NETWORK
TITLE = Betriebsmeldung
      A     #io_Ausgang_Motor;
      A     #in_Eingang_Motor;
      =     #io_Motor_in_Betrieb;
NETWORK
TITLE = Diskrepanz feststellen
      A     #io_Ausgang_Motor;
      AN    #in_Eingang_Motor;
      O;
      A     #in_Eingang_Motor;
      AN    #io_Ausgang_Motor;
      =     #Diskrepanz;
NETWORK
TITLE = Störungszähler
      A     #in_Quitt_Stoerung_noetig;
      AN    #in_Quitt_Stoerung;
      A     #io_Stoerung;
      O;
      A     #Diskrepanz;
      AN    #in_Quitt_Stoerung;	// (009)
      O;	// (009)
      AN    #in_Quitt_Stoerung_noetig;	// (009)
      A     #Diskrepanz;	// (009)
      JC    SZ1;
      L     0;	// Wenn keine Diskrepanz dann Zähler löschen
      T     DIW [AR2,P#6.0];	// Istzeit Störung (Struktur)
      JU    ESZ;
// Störungszähler in jeder Sekunde erhöhen
SZ1:  O     #io_Stoerung;
      ON    "M4.5 ImpulseClock1,0Sec";	// Sekundenimpuls (Standardmerker)
      JC    ESZ;
      L     DIW [AR2,P#6.0];	// Istzeit Störung (Struktur)
      INC   1;
      T     DIW [AR2,P#6.0];	// Istzeit Störung (Struktur)
ESZ:  NOP   0;
NETWORK
TITLE = Störmeldung ausgeben
      L     DIW [AR2,P#6.0];	// Istzeit Störung (Struktur)
      L     DIW [AR2,P#4.0];	// Sollzeit Störung (Struktur)
      >=I;
      =     #io_Stoerung;
NETWORK
TITLE = Stoerung quittieren
      O     #Diskrepanz;	// Stoerung steht noch an
      ON    #io_Stoerung;
      JC    ESQ;
      ON    #in_Quitt_Stoerung_noetig;	// Stoerung muß quittiert werden ?
      JC    SQ1;	// Stoerung muß nicht quittiert werden
      A     #in_Quitt_Stoerung;
SQ1:  R     #io_Stoerung;
ESQ:  NOP   0;
NETWORK
TITLE = Betriebsstundenzähler
//jede Sekunde wird der Sekundenzähler erhöht und beim erreichen von 3600 
//Sekunden wird eine Betriebsstunde addiert. (nur über Gleitpunktwert zu ungenau)
      ON    DIX [AR2,P#0.3];	// Kennung Betriebsstundenzähler ein (Struktur)
      ON    #io_Ausgang_Motor;
      ON    "M4.5 ImpulseClock1,0Sec";	// Sekundentakt
      JC    EBSZ;
      L     DIW [AR2,P#44.0];	// Betriebsstunden Sekundenzähler bis 3600 (007)
      L     1;	// (007)
      +I;	// (007)
      T     DIW [AR2,P#44.0];	// Betriebsstunden Sekundenzähler bis 3600 (007)
      L     3600;	// (007)
      <I;	// (007)
      JC    EBSZ;	// (007)
      L     DID [AR2,P#32.0];	// Betriebsstundenzähler (007)
      L     1.000000e+00;	// (007)
      +R;	// (007)
      T     DID [AR2,P#32.0];	// Betriebsstundenzähler (007)
      L     0;	// (007)
      T     DIW [AR2,P#44.0];	// Betriebsstunden Sekundenzähler bis 3600 (007)
EBSZ: NOP   0;
NETWORK
TITLE = Betriebsstundenzähler zurücksetzten
      AN    DIX [AR2,P#30.0];	// Reset Betriebsstundenzähler (Struktur)
      JC    E_RB;
      L     0.000000e+00;
      T     DID [AR2,P#32.0];	// Betriebsstundenzähler (Struktur)
      CLR;
      =     DIX [AR2,P#30.0];	// Reset Betriebsstundenzähler (Struktur)
E_RB: NOP   0;
NETWORK
TITLE = Warnmeldung Betriebsstundenzähler erzeugen
      A(;
      L     DID [AR2,P#32.0];	// Betriebsstundenzähler (Struktur)
      L     DID [AR2,P#36.0];	// Sollzeit Warnung (Struktur)
      >R;
      );
      A(;
      L     DID [AR2,P#36.0];	// Sollzeit Warnung (Struktur)
      L     0.000000e+00;
      <>R;
      );
      =     DIX [AR2,P#30.1];	// Warnmeldung Betriebsstundenzähler (Struktur)
NETWORK
TITLE = Alarmmeldung Betriebsstundenzähler erzeugen
      A(;
      L     DID [AR2,P#32.0];	// Betriebsstundenzähler (Struktur)
      L     DID [AR2,P#40.0];	// Sollzeit Alarm (Struktur)
      >R;
      );
      A(;
      L     DID [AR2,P#40.0];	// Sollzeit Alarm (Struktur)
      L     0.000000e+00;
      <>R;
      );
      =     DIX [AR2,P#30.2];	// Warnmeldung Betriebsstundenzähler (Struktur)
NETWORK
TITLE = Objektstatus für Visualisation OP // (011)(012)
//Stati:
//-------
//1 = nicht in Betrieb, keine Störung ==> Farborschlag weiß
//5 = angesteuert, in Betrieb, keine Störung ==> Farbvorschalg grün
//9 = angesteuert, nicht in Betrieb, keine Störung ==> Farbvorschalg grau
//16 = Störung ==> Farbvorschalg rot
// 1 = nicht in Betrieb, keine Störung ==> Farborschlag weiß
      L     1;
      AN    #io_Ausgang_Motor;
      AN    #in_Eingang_Motor;
      AN    #io_Stoerung;
      JC    disp;
// 5 = angesteuert, in Betrieb, keine Störung ==> Farbvorschalg grün
      L     5;
      A     #io_Ausgang_Motor;
      A     #in_Eingang_Motor;
      AN    #io_Stoerung;
      JC    disp;
// 9 = angesteuert, nicht in Betrieb, keine Störung ==> Farbvorschalg grau
      L     9;
      A     #io_Ausgang_Motor;
      AN    #in_Eingang_Motor;
      AN    #io_Stoerung;
      JC    disp;
// 16 = Störung ==> Farbvorschalg rot
      L     16;
      A     #io_Stoerung;
      JC    disp;
      L     0;
disp: T     #Objektstatus;
NETWORK
TITLE = Daten in Struktur speichern
      A     #in_Anlage_ein;	// (013)
      =     DIX [AR2,P#46.0];	// (013) Anlage ein (Struktur)
      A     #in_Eingang_Motor;
      =     DIX [AR2,P#2.1];	// Eingang Motor (Struktur)
      A     #io_Ausgang_Motor;
      =     DIX [AR2,P#2.0];	// Ausgang Motor (Struktur)
      A     #io_Motor_in_Betrieb;
      =     DIX [AR2,P#2.4];	// Motor in Betrieb (Struktur)
      A     #io_Stoerung;
      =     DIX [AR2,P#2.5];	// Störung (Struktur)
      A     #Taktanzahl_erreicht;
      =     DIX [AR2,P#3.3];	// Taktanzahl erreicht (Struktur)
      A     #Taktausgang;
      =     DIX [AR2,P#3.7];	// Taktausgang (Struktur)
      L     #Zeitzaehler;
      T     DID [AR2,P#16.0];	// Impuls-/Pausezähler (Struktur)
      L     #Taktzaehler;
      T     DIW [AR2,P#22.0];	// Taktzähler (Struktur)
      L     #Objektstatus;	// (011)
      T     DIW [AR2,P#48.0];	// #Objektstatus  (Struktur)   // (011)
NETWORK
TITLE = ENDE
      NOP   0;
END_FUNCTION

